Yaskawa INFORM job: A_ROOF_UPPER_0614_2_PAINT_11.JBI

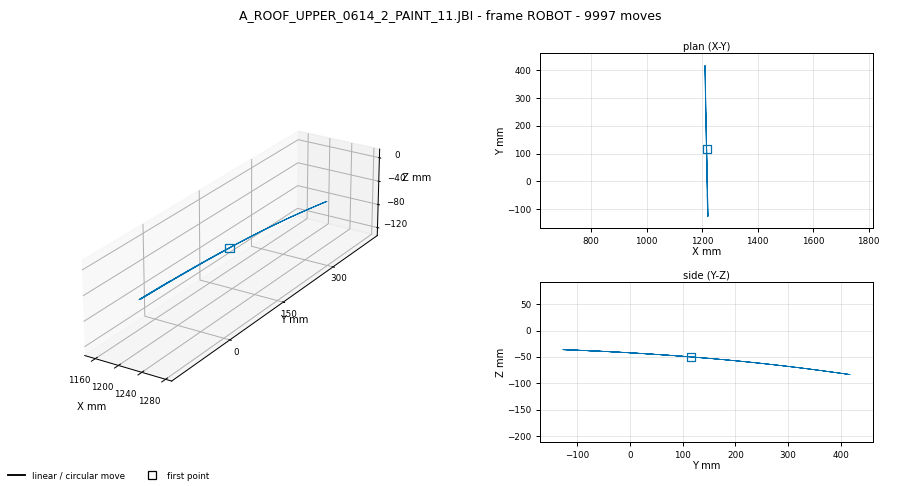
[picture p0: tool path of A_ROOF_UPPER_0614_2_PAINT_11.JBI in frame ROBOT, 9997 of 9997 moves have a stored position in this frame; points joined in program order, loops and branches not executed]
/JOB
//NAME A_ROOF_UPPER_0614_2_PAINT11
//POS
///NPOS 9997,0,0,0,0,0
///TOOL 1
///USER 0
///POSTYPE ROBOT
///RECTAN
///RCONF 1,0,0,0,0,0,0,0,0,0,0,0,0,0,0,0,0,0,0,0,0,0,0,0
C00000=1216.968,115.687,-49.725,-178.391,5.741,148.534
C00001=1216.973,115.438,-49.705,-178.393,5.741,148.535
C00002=1216.978,115.189,-49.686,-178.396,5.740,148.535
C00003=1216.982,114.939,-49.667,-178.398,5.738,148.536
C00004=1216.988,114.691,-49.647,-178.401,5.738,148.536
C00005=1216.992,114.441,-49.628,-178.403,5.737,148.537
C00006=1216.997,114.191,-49.608,-178.406,5.735,148.537
C00007=1217.002,113.943,-49.589,-178.408,5.734,148.538
C00008=1217.006,113.693,-49.570,-178.411,5.734,148.538
C00009=1217.012,113.445,-49.550,-178.414,5.732,148.539
C00010=1217.016,113.195,-49.531,-178.416,5.731,148.539
C00011=1217.020,112.946,-49.512,-178.419,5.731,148.540
C00012=1217.026,112.697,-49.492,-178.422,5.729,148.541
C00013=1217.031,112.447,-49.473,-178.424,5.728,148.541
C00014=1217.035,112.199,-49.454,-178.426,5.727,148.542
C00015=1217.040,111.949,-49.434,-178.430,5.726,148.542
C00016=1217.045,111.700,-49.415,-178.432,5.725,148.543
C00017=1217.049,111.451,-49.396,-178.434,5.724,148.543
C00018=1217.055,111.202,-49.377,-178.437,5.724,148.544
C00019=1217.060,110.952,-49.358,-178.440,5.722,148.544
C00020=1217.064,110.703,-49.339,-178.442,5.721,148.545
C00021=1217.069,110.454,-49.319,-178.444,5.720,148.545
C00022=1217.074,110.204,-49.300,-178.448,5.719,148.546
C00023=1217.078,109.956,-49.281,-178.450,5.718,148.546
C00024=1217.083,109.706,-49.261,-178.452,5.717,148.547
C00025=1217.088,109.457,-49.242,-178.455,5.716,148.547
C00026=1217.093,109.207,-49.224,-178.458,5.715,148.548
C00027=1217.098,108.959,-49.204,-178.460,5.714,148.549
C00028=1217.102,108.709,-49.185,-178.463,5.713,148.549
C00029=1217.107,108.460,-49.166,-178.466,5.712,148.550
C00030=1217.112,108.211,-49.146,-178.468,5.711,148.550
C00031=1217.117,107.962,-49.128,-178.470,5.710,148.551
C00032=1217.122,107.693,-49.107,-178.473,5.709,148.551
C00033=1217.128,107.425,-49.087,-178.476,5.708,148.552
C00034=1217.133,107.156,-49.066,-178.479,5.707,148.552
C00035=1217.138,106.888,-49.046,-178.481,5.706,148.553
C00036=1217.143,106.638,-49.027,-178.485,5.705,148.554
C00037=1217.147,106.389,-49.009,-178.487,5.704,148.554
C00038=1217.153,106.141,-48.989,-178.489,5.703,148.555
C00039=1217.157,105.891,-48.970,-178.492,5.701,148.555
C00040=1217.162,105.642,-48.952,-178.495,5.701,148.556
C00041=1217.167,105.392,-48.932,-178.497,5.700,148.556
C00042=1217.172,105.144,-48.913,-178.499,5.699,148.557
C00043=1217.177,104.893,-48.894,-178.503,5.698,148.558
C00044=1217.181,104.645,-48.876,-178.505,5.697,148.558
C00045=1217.186,104.395,-48.856,-178.507,5.696,148.559
C00046=1217.191,104.146,-48.838,-178.510,5.694,148.559
C00047=1217.195,103.898,-48.819,-178.513,5.694,148.560
C00048=1217.201,103.647,-48.800,-178.515,5.693,148.560
C00049=1217.205,103.399,-48.782,-178.517,5.692,148.561
C00050=1217.210,103.149,-48.762,-178.521,5.691,148.561
C00051=1217.215,102.900,-48.744,-178.523,5.690,148.562
C00052=1217.220,102.651,-48.724,-178.525,5.689,148.562
C00053=1217.224,102.401,-48.706,-178.528,5.689,148.563
C00054=1217.230,102.153,-48.687,-178.531,5.687,148.563
C00055=1217.234,101.903,-48.669,-178.533,5.686,148.564
C00056=1217.239,101.654,-48.649,-178.535,5.685,148.565
C00057=1217.244,101.405,-48.631,-178.538,5.685,148.565
C00058=1217.248,101.155,-48.612,-178.541,5.683,148.566
C00059=1217.254,100.906,-48.594,-178.543,5.682,148.566
C00060=1217.258,100.657,-48.575,-178.546,5.682,148.567
C00061=1217.264,100.407,-48.556,-178.549,5.680,148.568
C00062=1217.268,100.159,-48.537,-178.551,5.679,148.568
C00063=1217.273,99.909,-48.519,-178.554,5.679,148.569
C00064=1217.278,99.660,-48.500,-178.556,5.678,148.569
C00065=1217.283,99.411,-48.482,-178.559,5.676,148.570
C00066=1217.287,99.161,-48.463,-178.562,5.676,148.570
C00067=1217.292,98.912,-48.444,-178.564,5.675,148.571
C00068=1217.297,98.663,-48.426,-178.566,5.674,148.571
C00069=1217.301,98.413,-48.407,-178.569,5.672,148.572
C00070=1217.307,98.164,-48.389,-178.572,5.672,148.572
C00071=1217.312,97.915,-48.370,-178.574,5.671,148.573
C00072=1217.316,97.666,-48.352,-178.577,5.670,148.573
C00073=1217.321,97.417,-48.332,-178.579,5.670,148.574
C00074=1217.326,97.168,-48.314,-178.582,5.668,148.575
C00075=1217.331,96.918,-48.296,-178.584,5.667,148.575
C00076=1217.336,96.669,-48.277,-178.587,5.667,148.576
C00077=1217.341,96.420,-48.259,-178.589,5.666,148.576
C00078=1217.345,96.170,-48.240,-178.592,5.664,148.577
C00079=1217.350,95.921,-48.222,-178.595,5.664,148.578
C00080=1217.355,95.672,-48.203,-178.597,5.663,148.578
C00081=1217.360,95.422,-48.185,-178.600,5.662,148.579
C00082=1217.364,95.173,-48.166,-178.603,5.661,148.579
C00083=1217.370,94.924,-48.147,-178.605,5.660,148.580
C00084=1217.375,94.675,-48.129,-178.608,5.659,148.580
C00085=1217.379,94.425,-48.111,-178.610,5.659,148.581
C00086=1217.384,94.176,-48.092,-178.612,5.658,148.581
C00087=1217.389,93.927,-48.074,-178.616,5.656,148.582
C00088=1217.394,93.677,-48.056,-178.618,5.656,148.583
C00089=1217.399,93.428,-48.038,-178.620,5.655,148.583
C00090=1217.403,93.179,-48.019,-178.623,5.654,148.584
C00091=1217.408,92.930,-48.001,-178.626,5.652,148.584
C00092=1217.414,92.680,-47.982,-178.628,5.652,148.585
C00093=1217.418,92.430,-47.964,-178.631,5.651,148.585
C00094=1217.423,92.181,-47.946,-178.633,5.650,148.586
C00095=1217.428,91.933,-47.927,-178.636,5.650,148.587
C00096=1217.433,91.684,-47.909,-178.639,5.648,148.587
C00097=1217.437,91.434,-47.891,-178.641,5.647,148.588
C00098=1217.442,91.184,-47.872,-178.644,5.647,148.588
C00099=1217.447,90.935,-47.854,-178.646,5.646,148.589
C00100=1217.452,90.686,-47.836,-178.648,5.645,148.589
C00101=1217.457,90.437,-47.818,-178.652,5.644,148.590
C00102=1217.461,90.187,-47.799,-178.654,5.643,148.591
C00103=1217.466,89.938,-47.781,-178.656,5.642,148.591
C00104=1217.471,89.689,-47.763,-178.659,5.642,148.592
C00105=1217.476,89.440,-47.745,-178.662,5.641,148.592
C00106=1217.482,89.190,-47.727,-178.664,5.639,148.593
C00107=1217.486,88.941,-47.709,-178.667,5.639,148.593
C00108=1217.491,88.691,-47.691,-178.670,5.638,148.594
C00109=1217.496,88.442,-47.673,-178.672,5.637,148.594
C00110=1217.501,88.193,-47.655,-178.674,5.637,148.595
C00111=1217.506,87.944,-47.637,-178.677,5.635,148.596
C00112=1217.510,87.695,-47.619,-178.680,5.634,148.596
C00113=1217.515,87.445,-47.600,-178.682,5.634,148.597
C00114=1217.520,87.196,-47.582,-178.685,5.633,148.598
C00115=1217.525,86.946,-47.564,-178.687,5.632,148.598
C00116=1217.530,86.697,-47.546,-178.690,5.631,148.599
C00117=1217.534,86.448,-47.528,-178.693,5.630,148.599
C00118=1217.539,86.199,-47.510,-178.695,5.629,148.600
C00119=1217.544,85.949,-47.492,-178.698,5.629,148.600
C00120=1217.549,85.700,-47.474,-178.700,5.628,148.601
C00121=1217.553,85.451,-47.456,-178.702,5.627,148.601
C00122=1217.558,85.202,-47.438,-178.705,5.626,148.602
C00123=1217.563,84.952,-47.420,-178.708,5.625,148.603
C00124=1217.568,84.703,-47.402,-178.711,5.625,148.603
C00125=1217.573,84.454,-47.384,-178.713,5.624,148.604
C00126=1217.578,84.205,-47.366,-178.715,5.623,148.604
C00127=1217.583,83.956,-47.348,-178.718,5.622,148.605
C00128=1217.587,83.706,-47.330,-178.721,5.621,148.606
C00129=1217.592,83.456,-47.313,-178.723,5.620,148.606
C00130=1217.597,83.207,-47.295,-178.726,5.620,148.607
C00131=1217.602,82.958,-47.277,-178.728,5.619,148.607
C00132=1217.607,82.708,-47.259,-178.731,5.618,148.608
C00133=1217.612,82.459,-47.241,-178.733,5.617,148.609
C00134=1217.617,82.210,-47.223,-178.736,5.616,148.609
C00135=1217.622,81.960,-47.205,-178.739,5.615,148.610
C00136=1217.627,81.692,-47.186,-178.741,5.615,148.610
C00137=1217.632,81.424,-47.167,-178.744,5.614,148.611
C00138=1217.638,81.156,-47.147,-178.747,5.613,148.612
C00139=1217.643,80.887,-47.128,-178.750,5.612,148.612
C00140=1217.648,80.637,-47.111,-178.752,5.611,148.613
C00141=1217.653,80.388,-47.093,-178.755,5.610,148.613
C00142=1217.658,80.139,-47.075,-178.757,5.610,148.614
C00143=1217.663,79.889,-47.057,-178.760,5.608,148.615
C00144=1217.667,79.640,-47.040,-178.763,5.608,148.615
C00145=1217.672,79.391,-47.022,-178.765,5.607,148.616
C00146=1217.677,79.141,-47.005,-178.768,5.606,148.616
C00147=1217.682,78.892,-46.987,-178.770,5.605,148.617
C00148=1217.687,78.643,-46.969,-178.773,5.605,148.617
C00149=1217.692,78.394,-46.951,-178.775,5.604,148.618
C00150=1217.697,78.144,-46.933,-178.778,5.603,148.619
C00151=1217.701,77.895,-46.916,-178.781,5.602,148.619
C00152=1217.706,77.646,-46.898,-178.783,5.601,148.620
C00153=1217.711,77.396,-46.881,-178.786,5.601,148.620
C00154=1217.716,77.147,-46.863,-178.788,5.600,148.621
C00155=1217.721,76.898,-46.845,-178.791,5.599,148.622
C00156=1217.726,76.649,-46.828,-178.793,5.599,148.622
C00157=1217.731,76.399,-46.810,-178.796,5.598,148.623
C00158=1217.736,76.150,-46.793,-178.798,5.596,148.623
C00159=1217.741,75.900,-46.775,-178.801,5.596,148.624
C00160=1217.746,75.651,-46.757,-178.804,5.595,148.625
C00161=1217.750,75.402,-46.740,-178.806,5.595,148.625
C00162=1217.755,75.153,-46.722,-178.809,5.594,148.626
C00163=1217.760,74.903,-46.705,-178.811,5.593,148.626
C00164=1217.765,74.654,-46.687,-178.814,5.593,148.627
C00165=1217.770,74.404,-46.670,-178.816,5.592,148.627
C00166=1217.775,74.155,-46.652,-178.819,5.590,148.628
C00167=1217.779,73.906,-46.634,-178.822,5.590,148.629
C00168=1217.785,73.656,-46.617,-178.824,5.589,148.629
C00169=1217.789,73.407,-46.600,-178.826,5.588,148.630
C00170=1217.794,73.157,-46.583,-178.829,5.588,148.631
C00171=1217.800,72.909,-46.565,-178.832,5.587,148.631
C00172=1217.804,72.659,-46.548,-178.834,5.586,148.632
C00173=1217.809,72.410,-46.530,-178.837,5.585,148.632
C00174=1217.814,72.160,-46.513,-178.839,5.585,148.633
C00175=1217.819,71.911,-46.496,-178.842,5.584,148.634
C00176=1217.824,71.662,-46.478,-178.845,5.583,148.634
C00177=1217.829,71.412,-46.461,-178.847,5.582,148.635
C00178=1217.833,71.163,-46.444,-178.850,5.581,148.635
C00179=1217.838,70.913,-46.426,-178.852,5.581,148.636
C00180=1217.843,70.664,-46.408,-178.855,5.580,148.637
C00181=1217.848,70.415,-46.392,-178.857,5.579,148.637
C00182=1217.853,70.165,-46.375,-178.860,5.579,148.638
C00183=1217.858,69.916,-46.357,-178.862,5.578,148.638
C00184=1217.863,69.667,-46.340,-178.865,5.578,148.639
C00185=1217.868,69.418,-46.322,-178.867,5.577,148.640
C00186=1217.873,69.168,-46.305,-178.870,5.575,148.640
C00187=1217.877,68.918,-46.288,-178.873,5.575,148.641
C00188=1217.882,68.669,-46.270,-178.876,5.574,148.641
C00189=1217.887,68.420,-46.254,-178.878,5.573,148.642
C00190=1217.893,68.171,-46.237,-178.880,5.573,148.643
C00191=1217.897,67.922,-46.219,-178.883,5.572,148.643
C00192=1217.902,67.672,-46.202,-178.886,5.572,148.644
C00193=1217.907,67.422,-46.185,-178.888,5.571,148.644
C00194=1217.911,67.173,-46.168,-178.890,5.570,148.645
C00195=1217.917,66.923,-46.150,-178.893,5.569,148.646
C00196=1217.922,66.675,-46.134,-178.896,5.569,148.646
C00197=1217.927,66.426,-46.116,-178.898,5.568,148.647
C00198=1217.931,66.176,-46.099,-178.901,5.567,148.647
C00199=1217.936,65.926,-46.082,-178.904,5.566,148.648
C00200=1217.941,65.677,-46.065,-178.906,5.565,148.649
C00201=1217.946,65.428,-46.047,-178.909,5.565,148.649
C00202=1217.951,65.179,-46.031,-178.911,5.564,148.650
C00203=1217.956,64.929,-46.014,-178.914,5.563,148.650
C00204=1217.961,64.680,-45.997,-178.916,5.563,148.651
C00205=1217.966,64.430,-45.980,-178.919,5.562,148.652
C00206=1217.970,64.181,-45.962,-178.921,5.561,148.652
C00207=1217.976,63.932,-45.946,-178.924,5.561,148.653
C00208=1217.980,63.682,-45.929,-178.926,5.560,148.654
C00209=1217.985,63.432,-45.912,-178.929,5.560,148.654
C00210=1217.990,63.183,-45.895,-178.931,5.559,148.655
C00211=1217.996,62.934,-45.878,-178.934,5.558,148.655
C00212=1218.000,62.685,-45.861,-178.936,5.558,148.656
C00213=1218.005,62.435,-45.843,-178.939,5.557,148.657
C00214=1218.010,62.186,-45.827,-178.942,5.556,148.657
C00215=1218.015,61.936,-45.810,-178.944,5.555,148.658
C00216=1218.020,61.687,-45.793,-178.947,5.554,148.658
C00217=1218.024,61.438,-45.777,-178.950,5.554,148.659
C00218=1218.030,61.188,-45.759,-178.952,5.553,148.660
C00219=1218.034,60.938,-45.743,-178.955,5.552,148.660
C00220=1218.040,60.689,-45.726,-178.957,5.551,148.661
C00221=1218.044,60.440,-45.709,-178.960,5.551,148.662
C00222=1218.049,60.191,-45.691,-178.962,5.550,148.662
C00223=1218.054,59.942,-45.675,-178.965,5.550,148.663
C00224=1218.059,59.692,-45.658,-178.967,5.549,148.663
C00225=1218.064,59.443,-45.641,-178.970,5.548,148.664
C00226=1218.069,59.193,-45.624,-178.972,5.548,148.665
C00227=1218.074,58.944,-45.608,-178.975,5.547,148.665
C00228=1218.079,58.695,-45.591,-178.978,5.547,148.666
C00229=1218.083,58.445,-45.574,-178.980,5.546,148.666
C00230=1218.089,58.196,-45.557,-178.982,5.545,148.667
C00231=1218.094,57.946,-45.540,-178.985,5.545,148.668
C00232=1218.098,57.697,-45.524,-178.988,5.544,148.668
C00233=1218.104,57.448,-45.507,-178.990,5.543,148.669
C00234=1218.108,57.198,-45.490,-178.992,5.543,148.670
C00235=1218.113,56.948,-45.474,-178.995,5.542,148.670
C00236=1218.118,56.699,-45.457,-178.998,5.541,148.671
C00237=1218.123,56.450,-45.441,-179.000,5.541,148.672
C00238=1218.128,56.200,-45.424,-179.003,5.540,148.672
C00239=1218.132,55.951,-45.407,-179.005,5.539,148.673
C00240=1218.138,55.683,-45.389,-179.008,5.538,148.673
C00241=1218.144,55.415,-45.371,-179.011,5.537,148.674
C00242=1218.149,55.146,-45.354,-179.014,5.537,148.675
C00243=1218.155,54.877,-45.335,-179.016,5.536,148.675
C00244=1218.159,54.628,-45.319,-179.019,5.536,148.676
C00245=1218.164,54.378,-45.302,-179.022,5.535,148.677
C00246=1218.169,54.129,-45.285,-179.024,5.535,148.677
C00247=1218.174,53.879,-45.269,-179.027,5.534,148.678
C00248=1218.179,53.630,-45.253,-179.029,5.533,148.679
C00249=1218.184,53.381,-45.236,-179.032,5.533,148.679
C00250=1218.189,53.131,-45.219,-179.034,5.532,148.680
C00251=1218.194,52.882,-45.203,-179.037,5.531,148.680
C00252=1218.199,52.633,-45.186,-179.039,5.531,148.681
C00253=1218.203,52.383,-45.170,-179.042,5.530,148.682
C00254=1218.208,52.134,-45.154,-179.044,5.529,148.682
C00255=1218.214,51.884,-45.137,-179.047,5.529,148.683
C00256=1218.219,51.635,-45.120,-179.050,5.528,148.683
C00257=1218.223,51.385,-45.104,-179.052,5.528,148.684
C00258=1218.228,51.136,-45.088,-179.055,5.527,148.685
C00259=1218.233,50.887,-45.071,-179.057,5.527,148.686
C00260=1218.238,50.638,-45.055,-179.060,5.526,148.686
C00261=1218.244,50.388,-45.038,-179.062,5.525,148.687
C00262=1218.248,50.138,-45.022,-179.065,5.525,148.687
C00263=1218.253,49.889,-45.005,-179.067,5.524,148.688
C00264=1218.258,49.639,-44.990,-179.070,5.523,148.689
C00265=1218.262,49.390,-44.973,-179.072,5.523,148.689
C00266=1218.268,49.141,-44.957,-179.075,5.522,148.690
C00267=1218.272,48.892,-44.940,-179.078,5.521,148.690
C00268=1218.278,48.642,-44.924,-179.080,5.521,148.691
C00269=1218.283,48.393,-44.907,-179.083,5.520,148.692
C00270=1218.288,48.144,-44.891,-179.085,5.520,148.692
C00271=1218.293,47.894,-44.875,-179.088,5.519,148.693
C00272=1218.297,47.644,-44.858,-179.090,5.518,148.694
C00273=1218.302,47.395,-44.843,-179.093,5.518,148.694
C00274=1218.307,47.145,-44.826,-179.096,5.517,148.695
C00275=1218.312,46.897,-44.810,-179.098,5.517,148.696
C00276=1218.317,46.646,-44.794,-179.101,5.516,148.696
C00277=1218.322,46.398,-44.777,-179.103,5.515,148.697
C00278=1218.327,46.148,-44.761,-179.106,5.515,148.697
C00279=1218.332,45.898,-44.744,-179.108,5.514,148.698
C00280=1218.337,45.649,-44.728,-179.111,5.514,148.699
C00281=1218.342,45.400,-44.712,-179.114,5.513,148.699
C00282=1218.347,45.150,-44.696,-179.116,5.512,148.700
C00283=1218.352,44.901,-44.680,-179.118,5.512,148.700
C00284=1218.357,44.651,-44.663,-179.121,5.511,148.701
C00285=1218.362,44.402,-44.648,-179.124,5.510,148.702
C00286=1218.366,44.152,-44.631,-179.126,5.510,148.702
C00287=1218.372,43.903,-44.615,-179.129,5.509,148.703
C00288=1218.376,43.653,-44.599,-179.131,5.509,148.704
C00289=1218.382,43.404,-44.583,-179.134,5.508,148.704
C00290=1218.386,43.155,-44.567,-179.136,5.507,148.705
C00291=1218.392,42.905,-44.551,-179.139,5.507,148.706
C00292=1218.397,42.656,-44.535,-179.141,5.507,148.706
C00293=1218.401,42.406,-44.519,-179.144,5.506,148.707
C00294=1218.407,42.157,-44.503,-179.146,5.506,148.708
C00295=1218.411,41.907,-44.486,-179.149,5.505,148.708
C00296=1218.417,41.658,-44.471,-179.151,5.504,148.709
C00297=1218.421,41.408,-44.454,-179.154,5.504,148.709
C00298=1218.427,41.159,-44.439,-179.156,5.503,148.710
C00299=1218.430,40.910,-44.422,-179.159,5.503,148.711
C00300=1218.436,40.660,-44.407,-179.162,5.502,148.711
C00301=1218.441,40.411,-44.391,-179.164,5.502,148.712
C00302=1218.446,40.162,-44.375,-179.167,5.501,148.713
C00303=1218.451,39.912,-44.359,-179.169,5.500,148.713
C00304=1218.456,39.662,-44.343,-179.172,5.500,148.714
C00305=1218.461,39.413,-44.327,-179.174,5.499,148.715
C00306=1218.466,39.164,-44.311,-179.177,5.499,148.715
C00307=1218.471,38.914,-44.295,-179.180,5.498,148.716
C00308=1218.476,38.665,-44.279,-179.182,5.498,148.717
C00309=1218.481,38.415,-44.263,-179.185,5.497,148.717
C00310=1218.486,38.166,-44.248,-179.187,5.496,148.718
C00311=1218.491,37.917,-44.232,-179.189,5.496,148.718
C00312=1218.495,37.667,-44.216,-179.192,5.496,148.719
C00313=1218.501,37.418,-44.200,-179.194,5.495,148.720
C00314=1218.505,37.168,-44.183,-179.197,5.495,148.720
C00315=1218.511,36.919,-44.168,-179.200,5.494,148.721
C00316=1218.516,36.669,-44.152,-179.202,5.494,148.722
C00317=1218.520,36.419,-44.137,-179.205,5.493,148.722
C00318=1218.525,36.171,-44.121,-179.207,5.492,148.723
C00319=1218.531,35.921,-44.105,-179.210,5.492,148.724
C00320=1218.535,35.671,-44.089,-179.212,5.491,148.724
C00321=1218.541,35.422,-44.074,-179.215,5.491,148.725
C00322=1218.546,35.173,-44.057,-179.218,5.490,148.726
C00323=1218.550,34.923,-44.042,-179.220,5.489,148.726
C00324=1218.555,34.674,-44.026,-179.223,5.489,148.727
C00325=1218.561,34.424,-44.011,-179.225,5.489,148.727
C00326=1218.565,34.174,-43.995,-179.227,5.488,148.728
C00327=1218.571,33.925,-43.979,-179.230,5.488,148.729
C00328=1218.575,33.676,-43.963,-179.232,5.487,148.729
C00329=1218.580,33.426,-43.947,-179.235,5.487,148.730
C00330=1218.585,33.177,-43.932,-179.238,5.486,148.731
C00331=1218.591,32.927,-43.916,-179.240,5.486,148.731
C00332=1218.595,32.678,-43.901,-179.243,5.485,148.732
C00333=1218.600,32.428,-43.885,-179.245,5.484,148.733
C00334=1218.606,32.179,-43.870,-179.248,5.484,148.733
C00335=1218.610,31.929,-43.853,-179.250,5.483,148.734
C00336=1218.615,31.680,-43.838,-179.253,5.483,148.735
C00337=1218.620,31.431,-43.823,-179.255,5.483,148.735
C00338=1218.625,31.182,-43.807,-179.258,5.482,148.736
C00339=1218.629,30.932,-43.792,-179.260,5.482,148.737
C00340=1218.635,30.682,-43.776,-179.263,5.481,148.737
C00341=1218.640,30.433,-43.760,-179.266,5.481,148.738
C00342=1218.644,30.183,-43.745,-179.268,5.480,148.738
C00343=1218.650,29.934,-43.729,-179.271,5.479,148.739
C00344=1218.655,29.665,-43.712,-179.273,5.479,148.740
C00345=1218.661,29.397,-43.695,-179.276,5.478,148.741
C00346=1218.666,29.128,-43.680,-179.279,5.478,148.741
C00347=1218.671,28.859,-43.663,-179.282,5.477,148.742
C00348=1218.676,28.609,-43.647,-179.284,5.477,148.743
C00349=1218.681,28.360,-43.632,-179.286,5.476,148.743
C00350=1218.686,28.111,-43.616,-179.289,5.475,148.744
C00351=1218.692,27.861,-43.601,-179.292,5.475,148.745
C00352=1218.696,27.612,-43.586,-179.294,5.475,148.745
C00353=1218.701,27.362,-43.570,-179.296,5.475,148.746
C00354=1218.707,27.113,-43.554,-179.299,5.474,148.747
C00355=1218.711,26.864,-43.539,-179.302,5.473,148.747
C00356=1218.717,26.614,-43.523,-179.304,5.473,148.748
C00357=1218.721,26.365,-43.508,-179.307,5.472,148.749
C00358=1218.726,26.115,-43.493,-179.310,5.472,148.749
C00359=1218.732,25.865,-43.478,-179.312,5.471,148.750
C00360=1218.736,25.616,-43.463,-179.314,5.470,148.750
C00361=1218.742,25.367,-43.447,-179.317,5.471,148.751
C00362=1218.746,25.117,-43.432,-179.319,5.470,148.752
C00363=1218.751,24.867,-43.416,-179.322,5.470,148.752
C00364=1218.756,24.618,-43.401,-179.324,5.469,148.753
C00365=1218.761,24.369,-43.386,-179.327,5.469,148.754
C00366=1218.767,24.119,-43.371,-179.330,5.468,148.755
C00367=1218.771,23.869,-43.355,-179.332,5.468,148.755
C00368=1218.776,23.620,-43.340,-179.335,5.467,148.756
C00369=1218.781,23.371,-43.325,-179.337,5.467,148.756
C00370=1218.786,23.121,-43.309,-179.339,5.466,148.757
C00371=1218.791,22.872,-43.294,-179.342,5.466,148.758
C00372=1218.797,22.622,-43.279,-179.345,5.465,148.758
C00373=1218.801,22.372,-43.264,-179.347,5.465,148.759
C00374=1218.806,22.123,-43.248,-179.350,5.464,148.760
C00375=1218.811,21.874,-43.233,-179.352,5.464,148.760
C00376=1218.816,21.624,-43.218,-179.355,5.464,148.761
C00377=1218.821,21.375,-43.203,-179.357,5.463,148.762
C00378=1218.827,21.125,-43.188,-179.360,5.463,148.762
C00379=1218.831,20.876,-43.173,-179.362,5.462,148.763
C00380=1218.837,20.626,-43.158,-179.365,5.461,148.764
C00381=1218.841,20.376,-43.143,-179.367,5.461,148.764
C00382=1218.846,20.127,-43.127,-179.370,5.460,148.765
C00383=1218.851,19.878,-43.112,-179.372,5.461,148.766
C00384=1218.856,19.628,-43.098,-179.375,5.460,148.766
C00385=1218.861,19.379,-43.082,-179.377,5.460,148.767
C00386=1218.866,19.130,-43.067,-179.380,5.459,148.768
C00387=1218.872,18.880,-43.052,-179.383,5.459,148.768
C00388=1218.876,18.631,-43.037,-179.385,5.458,148.769
C00389=1218.882,18.381,-43.022,-179.388,5.458,148.770
C00390=1218.886,18.131,-43.007,-179.389,5.457,148.770
C00391=1218.891,17.882,-42.992,-179.392,5.457,148.771
C00392=1218.896,17.632,-42.977,-179.395,5.456,148.772
C00393=1218.901,17.383,-42.962,-179.397,5.456,148.772
C00394=1218.906,17.133,-42.947,-179.400,5.455,148.773
C00395=1218.911,16.884,-42.932,-179.403,5.455,148.774
C00396=1218.916,16.634,-42.917,-179.405,5.454,148.774
C00397=1218.921,16.385,-42.902,-179.407,5.455,148.775
C00398=1218.926,16.135,-42.888,-179.410,5.454,148.776
C00399=1218.932,15.886,-42.872,-179.413,5.453,148.776
C00400=1218.936,15.637,-42.857,-179.415,5.453,148.777
C00401=1218.941,15.387,-42.843,-179.418,5.452,148.778
C00402=1218.947,15.138,-42.827,-179.420,5.452,148.778
C00403=1218.952,14.888,-42.813,-179.422,5.452,148.779
C00404=1218.956,14.639,-42.798,-179.425,5.451,148.780
C00405=1218.962,14.389,-42.783,-179.428,5.451,148.780
C00406=1218.966,14.139,-42.768,-179.430,5.450,148.781
C00407=1218.971,13.889,-42.753,-179.433,5.450,148.782
C00408=1218.976,13.640,-42.738,-179.436,5.449,148.782
C00409=1218.981,13.390,-42.723,-179.438,5.449,148.783
C00410=1218.986,13.141,-42.708,-179.440,5.449,148.784
C00411=1218.991,12.891,-42.694,-179.443,5.448,148.784
C00412=1218.996,12.642,-42.679,-179.446,5.448,148.785
C00413=1219.001,12.392,-42.664,-179.448,5.447,148.786
C00414=1219.006,12.143,-42.649,-179.451,5.447,148.786
C00415=1219.012,11.893,-42.634,-179.452,5.447,148.787
C00416=1219.016,11.644,-42.619,-179.455,5.446,148.787
C00417=1219.021,11.394,-42.605,-179.458,5.446,148.788
C00418=1219.026,11.145,-42.590,-179.460,5.445,148.789
C00419=1219.032,10.895,-42.575,-179.463,5.445,148.790
C00420=1219.037,10.646,-42.561,-179.465,5.445,148.790
C00421=1219.041,10.397,-42.546,-179.468,5.444,148.791
C00422=1219.047,10.148,-42.532,-179.470,5.444,148.792
C00423=1219.052,9.898,-42.517,-179.473,5.443,148.792
C00424=1219.057,9.648,-42.502,-179.476,5.443,148.793
C00425=1219.062,9.399,-42.488,-179.478,5.443,148.794
C00426=1219.067,9.150,-42.473,-179.480,5.443,148.794
C00427=1219.072,8.900,-42.459,-179.483,5.442,148.795
C00428=1219.077,8.650,-42.444,-179.486,5.442,148.796
C00429=1219.082,8.401,-42.429,-179.488,5.441,148.796
C00430=1219.087,8.151,-42.415,-179.491,5.440,148.797
C00431=1219.092,7.901,-42.400,-179.493,5.440,148.798
C00432=1219.097,7.652,-42.385,-179.495,5.440,148.798
C00433=1219.102,7.402,-42.370,-179.498,5.439,148.799
C00434=1219.107,7.153,-42.356,-179.501,5.439,148.800
C00435=1219.112,6.903,-42.341,-179.503,5.438,148.800
C00436=1219.117,6.654,-42.327,-179.505,5.439,148.801
C00437=1219.122,6.404,-42.313,-179.508,5.438,148.802
C00438=1219.127,6.154,-42.298,-179.511,5.438,148.802
C00439=1219.132,5.906,-42.284,-179.513,5.437,148.803
C00440=1219.138,5.656,-42.269,-179.516,5.437,148.804
C00441=1219.143,5.406,-42.255,-179.518,5.437,148.804
C00442=1219.148,5.156,-42.240,-179.521,5.436,148.805
C00443=1219.152,4.907,-42.225,-179.523,5.436,148.806
C00444=1219.157,4.658,-42.211,-179.526,5.435,148.806
C00445=1219.162,4.408,-42.197,-179.528,5.434,148.807
C00446=1219.167,4.158,-42.182,-179.530,5.435,148.808
C00447=1219.172,3.909,-42.167,-179.533,5.434,148.808
C00448=1219.178,3.639,-42.152,-179.536,5.434,148.809
C00449=1219.184,3.371,-42.137,-179.539,5.434,148.810
C00450=1219.189,3.103,-42.121,-179.541,5.433,148.811
C00451=1219.194,2.833,-42.106,-179.544,5.433,148.811
C00452=1219.199,2.583,-42.092,-179.547,5.432,148.812
C00453=1219.204,2.334,-42.077,-179.549,5.432,148.813
C00454=1219.209,2.085,-42.062,-179.551,5.432,148.813
C00455=1219.214,1.835,-42.048,-179.554,5.431,148.814
C00456=1219.219,1.586,-42.034,-179.557,5.431,148.815
C00457=1219.224,1.336,-42.020,-179.559,5.430,148.815
C00458=1219.229,1.086,-42.006,-179.561,5.431,148.816
C00459=1219.234,0.837,-41.991,-179.564,5.430,148.817
C00460=1219.240,0.587,-41.976,-179.567,5.430,148.817
C00461=1219.244,0.338,-41.961,-179.569,5.429,148.818
C00462=1219.250,0.089,-41.947,-179.571,5.429,148.819
C00463=1219.255,-0.161,-41.933,-179.574,5.428,148.819
C00464=1219.260,-0.411,-41.919,-179.576,5.428,148.820
C00465=1219.265,-0.660,-41.905,-179.579,5.427,148.821
C00466=1219.270,-0.910,-41.890,-179.581,5.427,148.821
C00467=1219.275,-1.160,-41.876,-179.584,5.427,148.822
C00468=1219.280,-1.409,-41.862,-179.586,5.427,148.823
C00469=1219.285,-1.658,-41.849,-179.589,5.426,148.823
C00470=1219.290,-1.908,-41.834,-179.592,5.426,148.824
C00471=1219.294,-2.158,-41.820,-179.594,5.426,148.825
C00472=1219.299,-2.407,-41.806,-179.596,5.425,148.826
C00473=1219.305,-2.656,-41.792,-179.599,5.425,148.826
C00474=1219.310,-2.906,-41.777,-179.602,5.424,148.827
C00475=1219.315,-3.156,-41.763,-179.604,5.425,148.828
C00476=1219.320,-3.406,-41.749,-179.606,5.424,148.828
C00477=1219.325,-3.655,-41.735,-179.609,5.424,148.829
C00478=1219.330,-3.904,-41.721,-179.612,5.423,148.830
C00479=1219.335,-4.154,-41.706,-179.614,5.423,148.830
C00480=1219.340,-4.404,-41.692,-179.616,5.423,148.831
C00481=1219.346,-4.653,-41.678,-179.618,5.422,148.831
C00482=1219.351,-4.902,-41.664,-179.621,5.422,148.832
C00483=1219.356,-5.152,-41.650,-179.623,5.422,148.833
C00484=1219.360,-5.402,-41.637,-179.626,5.421,148.834
C00485=1219.366,-5.651,-41.623,-179.629,5.421,148.834
C00486=1219.371,-5.901,-41.609,-179.631,5.420,148.835
C00487=1219.376,-6.151,-41.594,-179.633,5.421,148.836
C00488=1219.381,-6.400,-41.580,-179.636,5.420,148.836
C00489=1219.386,-6.649,-41.566,-179.639,5.420,148.837
C00490=1219.391,-6.899,-41.552,-179.641,5.419,148.838
C00491=1219.395,-7.148,-41.538,-179.643,5.419,148.838
C00492=1219.401,-7.399,-41.525,-179.646,5.419,148.839
C00493=1219.406,-7.648,-41.511,-179.649,5.418,148.840
C00494=1219.411,-7.897,-41.496,-179.651,5.418,148.840
C00495=1219.416,-8.147,-41.482,-179.653,5.418,148.841
C00496=1219.422,-8.396,-41.468,-179.656,5.418,148.842
C00497=1219.426,-8.646,-41.455,-179.659,5.417,148.843
C00498=1219.431,-8.896,-41.441,-179.661,5.417,148.843
C00499=1219.437,-9.145,-41.427,-179.663,5.417,148.844
C00500=1219.442,-9.395,-41.413,-179.666,5.416,148.845
C00501=1219.447,-9.644,-41.399,-179.669,5.416,148.845
C00502=1219.451,-9.894,-41.385,-179.671,5.415,148.846
C00503=1219.457,-10.143,-41.372,-179.673,5.415,148.846
C00504=1219.462,-10.393,-41.357,-179.676,5.415,148.847
C00505=1219.467,-10.643,-41.343,-179.678,5.414,148.848
C00506=1219.471,-10.891,-41.330,-179.681,5.414,148.849
C00507=1219.477,-11.142,-41.316,-179.683,5.414,148.849
C00508=1219.482,-11.392,-41.302,-179.686,5.414,148.850
C00509=1219.487,-11.641,-41.288,-179.688,5.413,148.851
C00510=1219.492,-11.891,-41.274,-179.691,5.413,148.851
C00511=1219.497,-12.140,-41.261,-179.693,5.413,148.852
C00512=1219.502,-12.389,-41.247,-179.696,5.412,148.853
C00513=1219.507,-12.640,-41.233,-179.698,5.412,148.853
C00514=1219.512,-12.888,-41.220,-179.700,5.412,148.854
C00515=1219.517,-13.138,-41.206,-179.703,5.412,148.855
C00516=1219.522,-13.388,-41.191,-179.706,5.411,148.855
C00517=1219.528,-13.637,-41.178,-179.708,5.411,148.856
C00518=1219.532,-13.887,-41.165,-179.710,5.411,148.857
C00519=1219.538,-14.137,-41.151,-179.713,5.411,148.858
C00520=1219.543,-14.386,-41.137,-179.716,5.410,148.858
C00521=1219.547,-14.636,-41.123,-179.718,5.410,148.859
C00522=1219.553,-14.885,-41.110,-179.721,5.410,148.860
C00523=1219.558,-15.135,-41.096,-179.723,5.409,148.860
C00524=1219.562,-15.384,-41.082,-179.726,5.409,148.861
C00525=1219.568,-15.634,-41.069,-179.728,5.409,148.862
C00526=1219.573,-15.884,-41.055,-179.731,5.409,148.862
C00527=1219.578,-16.133,-41.042,-179.733,5.408,148.863
C00528=1219.583,-16.383,-41.028,-179.736,5.408,148.864
C00529=1219.589,-16.633,-41.014,-179.738,5.408,148.865
C00530=1219.593,-16.882,-41.001,-179.740,5.407,148.865
C00531=1219.598,-17.131,-40.987,-179.743,5.407,148.866
C00532=1219.604,-17.381,-40.974,-179.745,5.407,148.866
C00533=1219.608,-17.630,-40.960,-179.748,5.406,148.867
C00534=1219.614,-17.880,-40.947,-179.750,5.406,148.868
C00535=1219.618,-18.129,-40.933,-179.753,5.405,148.868
C00536=1219.624,-18.380,-40.919,-179.755,5.406,148.869
C00537=1219.629,-18.629,-40.905,-179.758,5.405,148.870
C00538=1219.634,-18.879,-40.893,-179.760,5.405,148.871
C00539=1219.639,-19.128,-40.879,-179.762,5.405,148.871
C00540=1219.644,-19.378,-40.866,-179.765,5.405,148.872
C00541=1219.649,-19.627,-40.852,-179.768,5.404,148.873
C00542=1219.655,-19.877,-40.838,-179.770,5.404,148.873
C00543=1219.659,-20.126,-40.825,-179.772,5.404,148.874
C00544=1219.665,-20.376,-40.811,-179.775,5.403,148.875
C00545=1219.670,-20.625,-40.799,-179.778,5.403,148.875
C00546=1219.675,-20.875,-40.784,-179.780,5.403,148.876
C00547=1219.680,-21.125,-40.772,-179.782,5.403,148.877
C00548=1219.685,-21.374,-40.758,-179.785,5.402,148.877
C00549=1219.691,-21.624,-40.744,-179.787,5.403,148.878
C00550=1219.695,-21.873,-40.731,-179.790,5.402,148.879
C00551=1219.701,-22.123,-40.717,-179.792,5.402,148.880
C00552=1219.706,-22.392,-40.703,-179.795,5.401,148.880
C00553=1219.711,-22.662,-40.689,-179.797,5.401,148.881
C00554=1219.717,-22.931,-40.674,-179.800,5.401,148.882
C00555=1219.722,-23.200,-40.660,-179.803,5.401,148.883
C00556=1219.727,-23.450,-40.646,-179.806,5.400,148.883
C00557=1219.732,-23.699,-40.634,-179.808,5.401,148.884
C00558=1219.738,-23.950,-40.620,-179.810,5.400,148.885
C00559=1219.742,-24.199,-40.607,-179.813,5.399,148.885
C00560=1219.748,-24.449,-40.593,-179.815,5.400,148.886
C00561=1219.753,-24.698,-40.581,-179.817,5.399,148.887
C00562=1219.758,-24.948,-40.566,-179.820,5.399,148.887
C00563=1219.763,-25.197,-40.554,-179.823,5.398,148.888
C00564=1219.768,-25.448,-40.540,-179.825,5.398,148.889
C00565=1219.773,-25.696,-40.527,-179.827,5.398,148.889
C00566=1219.778,-25.946,-40.514,-179.830,5.397,148.890
C00567=1219.783,-26.196,-40.501,-179.832,5.398,148.891
C00568=1219.789,-26.445,-40.488,-179.835,5.397,148.891
C00569=1219.793,-26.695,-40.474,-179.837,5.397,148.892
C00570=1219.799,-26.944,-40.461,-179.840,5.397,148.893
C00571=1219.804,-27.195,-40.448,-179.842,5.397,148.893
C00572=1219.809,-27.444,-40.435,-179.845,5.396,148.894
C00573=1219.813,-27.693,-40.421,-179.847,5.396,148.895
C00574=1219.819,-27.943,-40.408,-179.850,5.396,148.896
C00575=1219.824,-28.193,-40.395,-179.852,5.395,148.896
C00576=1219.829,-28.443,-40.382,-179.854,5.396,148.897
C00577=1219.835,-28.692,-40.369,-179.857,5.395,148.898
C00578=1219.839,-28.941,-40.356,-179.860,5.395,148.898
C00579=1219.845,-29.191,-40.342,-179.862,5.395,148.899
C00580=1219.849,-29.441,-40.330,-179.864,5.395,148.900
C00581=1219.854,-29.690,-40.317,-179.867,5.394,148.900
C00582=1219.860,-29.940,-40.304,-179.869,5.394,148.901
C00583=1219.864,-30.189,-40.290,-179.872,5.394,148.902
C00584=1219.870,-30.439,-40.277,-179.874,5.393,148.903
C00585=1219.875,-30.689,-40.264,-179.877,5.394,148.903
C00586=1219.880,-30.938,-40.251,-179.879,5.393,148.904
C00587=1219.885,-31.188,-40.239,-179.882,5.393,148.905
C00588=1219.890,-31.438,-40.225,-179.884,5.393,148.905
C00589=1219.895,-31.687,-40.213,-179.887,5.393,148.906
C00590=1219.901,-31.936,-40.200,-179.889,5.392,148.907
C00591=1219.906,-32.187,-40.186,-179.891,5.392,148.907
C00592=1219.911,-32.436,-40.173,-179.894,5.392,148.908
C00593=1219.916,-32.685,-40.160,-179.897,5.391,148.909
C00594=1219.921,-32.935,-40.147,-179.898,5.391,148.909
C00595=1219.926,-33.184,-40.134,-179.901,5.391,148.910
C00596=1219.931,-33.435,-40.121,-179.904,5.390,148.911
C00597=1219.937,-33.684,-40.108,-179.906,5.391,148.911
C00598=1219.942,-33.933,-40.096,-179.908,5.390,148.912
C00599=1219.946,-34.183,-40.083,-179.911,5.390,148.913
C00600=1219.951,-34.433,-40.070,-179.913,5.390,148.914
C00601=1219.957,-34.682,-40.057,-179.916,5.390,148.914
C00602=1219.962,-34.932,-40.044,-179.918,5.389,148.915
C00603=1219.967,-35.182,-40.031,-179.920,5.389,148.916
C00604=1219.972,-35.431,-40.019,-179.923,5.389,148.916
C00605=1219.978,-35.681,-40.005,-179.925,5.389,148.917
C00606=1219.982,-35.931,-39.992,-179.928,5.389,148.918
C00607=1219.987,-36.180,-39.980,-179.931,5.388,148.918
C00608=1219.993,-36.429,-39.967,-179.933,5.389,148.919
C00609=1219.997,-36.679,-39.954,-179.935,5.388,148.920
C00610=1220.003,-36.929,-39.941,-179.938,5.388,148.920
C00611=1220.008,-37.178,-39.928,-179.940,5.388,148.921
C00612=1220.013,-37.428,-39.915,-179.943,5.388,148.922
C00613=1220.018,-37.678,-39.903,-179.945,5.387,148.923
C00614=1220.024,-37.927,-39.890,-179.947,5.387,148.923
C00615=1220.029,-38.177,-39.877,-179.950,5.387,148.924
C00616=1220.034,-38.427,-39.865,-179.953,5.386,148.925
C00617=1220.039,-38.677,-39.852,-179.955,5.387,148.925
C00618=1220.044,-38.926,-39.840,-179.958,5.386,148.926
C00619=1220.049,-39.175,-39.827,-179.960,5.386,148.927
C00620=1220.054,-39.426,-39.813,-179.962,5.386,148.927
C00621=1220.059,-39.675,-39.801,-179.965,5.386,148.928
C00622=1220.064,-39.924,-39.788,-179.967,5.386,148.929
C00623=1220.070,-40.173,-39.776,-179.970,5.385,148.930
C00624=1220.074,-40.424,-39.763,-179.972,5.385,148.930
C00625=1220.079,-40.673,-39.751,-179.974,5.385,148.931
C00626=1220.085,-40.923,-39.738,-179.977,5.385,148.932
C00627=1220.090,-41.172,-39.726,-179.980,5.384,148.932
C00628=1220.095,-41.422,-39.712,-179.982,5.385,148.933
C00629=1220.100,-41.672,-39.699,-179.984,5.384,148.934
C00630=1220.106,-41.922,-39.688,-179.986,5.384,148.934
C00631=1220.111,-42.171,-39.675,-179.989,5.384,148.935
C00632=1220.115,-42.421,-39.662,-179.991,5.383,148.936
C00633=1220.120,-42.670,-39.649,-179.994,5.384,148.936
C00634=1220.125,-42.920,-39.637,-179.996,5.383,148.937
C00635=1220.131,-43.170,-39.625,-179.999,5.383,148.938
C00636=1220.136,-43.419,-39.612,179.999,5.383,148.938
C00637=1220.140,-43.669,-39.599,179.996,5.382,148.939
C00638=1220.146,-43.918,-39.587,179.994,5.383,148.940
C00639=1220.152,-44.168,-39.574,179.992,5.382,148.941
C00640=1220.157,-44.418,-39.562,179.989,5.382,148.941
C00641=1220.162,-44.667,-39.549,179.987,5.382,148.942
C00642=1220.167,-44.917,-39.536,179.984,5.382,148.943
C00643=1220.172,-45.167,-39.524,179.982,5.381,148.943
C00644=1220.177,-45.416,-39.512,179.979,5.381,148.944
C00645=1220.182,-45.666,-39.499,179.977,5.381,148.945
C00646=1220.188,-45.916,-39.487,179.975,5.381,148.945
C00647=1220.193,-46.165,-39.475,179.972,5.381,148.946
C00648=1220.197,-46.415,-39.462,179.969,5.380,148.947
C00649=1220.203,-46.665,-39.450,179.967,5.381,148.948
C00650=1220.208,-46.914,-39.437,179.965,5.380,148.948
C00651=1220.213,-47.164,-39.424,179.962,5.380,148.949
C00652=1220.218,-47.413,-39.413,179.960,5.380,148.950
C00653=1220.224,-47.663,-39.400,179.957,5.380,148.950
C00654=1220.228,-47.913,-39.387,179.955,5.380,148.951
C00655=1220.233,-48.163,-39.375,179.953,5.379,148.952
C00656=1220.239,-48.432,-39.362,179.950,5.379,148.953
C00657=1220.244,-48.702,-39.349,179.948,5.379,148.953
C00658=1220.250,-48.972,-39.335,179.945,5.379,148.954
C00659=1220.256,-49.242,-39.322,179.942,5.379,148.955
C00660=1220.261,-49.491,-39.309,179.940,5.378,148.955
C00661=1220.266,-49.742,-39.297,179.938,5.378,148.956
C00662=1220.271,-49.991,-39.285,179.935,5.378,148.957
C00663=1220.277,-50.241,-39.273,179.933,5.378,148.957
C00664=1220.281,-50.490,-39.261,179.930,5.378,148.958
C00665=1220.286,-50.739,-39.248,179.928,5.377,148.959
C00666=1220.291,-50.989,-39.236,179.926,5.378,148.960
C00667=1220.297,-51.239,-39.224,179.923,5.377,148.960
C00668=1220.302,-51.489,-39.212,179.921,5.377,148.961
C00669=1220.307,-51.738,-39.199,179.918,5.377,148.962
C00670=1220.313,-51.988,-39.187,179.915,5.376,148.962
C00671=1220.317,-52.238,-39.174,179.913,5.377,148.963
C00672=1220.323,-52.488,-39.162,179.911,5.376,148.964
C00673=1220.328,-52.737,-39.150,179.909,5.377,148.964
C00674=1220.332,-52.987,-39.138,179.906,5.376,148.965
C00675=1220.337,-53.236,-39.126,179.903,5.376,148.966
C00676=1220.343,-53.486,-39.114,179.901,5.376,148.967
C00677=1220.348,-53.735,-39.101,179.898,5.376,148.967
C00678=1220.353,-53.985,-39.089,179.896,5.376,148.968
C00679=1220.359,-54.235,-39.077,179.894,5.375,148.969
C00680=1220.363,-54.484,-39.066,179.891,5.375,148.969
C00681=1220.369,-54.734,-39.054,179.889,5.375,148.970
C00682=1220.374,-54.983,-39.041,179.886,5.375,148.971
C00683=1220.379,-55.233,-39.029,179.884,5.375,148.972
C00684=1220.384,-55.483,-39.017,179.882,5.375,148.972
C00685=1220.390,-55.733,-39.005,179.879,5.374,148.973
C00686=1220.394,-55.983,-38.993,179.877,5.375,148.974
C00687=1220.399,-56.232,-38.980,179.874,5.374,148.974
C00688=1220.404,-56.482,-38.969,179.873,5.374,148.975
C00689=1220.410,-56.731,-38.956,179.870,5.374,148.976
C00690=1220.415,-56.981,-38.944,179.868,5.374,148.976
C00691=1220.420,-57.231,-38.933,179.865,5.373,148.977
C00692=1220.425,-57.480,-38.920,179.862,5.373,148.978
C00693=1220.430,-57.730,-38.908,179.860,5.373,148.978
C00694=1220.436,-57.980,-38.896,179.858,5.373,148.979
C00695=1220.440,-58.229,-38.884,179.856,5.373,148.980
C00696=1220.446,-58.479,-38.873,179.853,5.373,148.980
C00697=1220.451,-58.729,-38.861,179.850,5.372,148.981
C00698=1220.456,-58.978,-38.848,179.848,5.373,148.982
C00699=1220.461,-59.228,-38.837,179.846,5.372,148.983
C00700=1220.466,-59.478,-38.825,179.843,5.373,148.983
C00701=1220.471,-59.727,-38.812,179.841,5.372,148.984
C00702=1220.477,-59.977,-38.800,179.839,5.372,148.985
C00703=1220.481,-60.227,-38.789,179.836,5.372,148.985
C00704=1220.487,-60.477,-38.777,179.833,5.371,148.986
C00705=1220.492,-60.726,-38.765,179.831,5.372,148.987
C00706=1220.497,-60.976,-38.753,179.829,5.371,148.987
C00707=1220.502,-61.226,-38.741,179.827,5.372,148.988
C00708=1220.508,-61.475,-38.730,179.824,5.371,148.989
C00709=1220.513,-61.724,-38.718,179.822,5.372,148.990
C00710=1220.518,-61.974,-38.706,179.819,5.371,148.990
C00711=1220.523,-62.224,-38.694,179.816,5.371,148.991
C00712=1220.529,-62.474,-38.682,179.815,5.371,148.991
C00713=1220.533,-62.723,-38.670,179.812,5.370,148.992
C00714=1220.539,-62.973,-38.658,179.810,5.370,148.993
C00715=1220.544,-63.223,-38.646,179.807,5.370,148.994
C00716=1220.549,-63.472,-38.635,179.805,5.370,148.994
C00717=1220.554,-63.722,-38.623,179.803,5.370,148.995
C00718=1220.559,-63.972,-38.612,179.800,5.369,148.996
C00719=1220.564,-64.221,-38.599,179.798,5.370,148.996
C00720=1220.569,-64.471,-38.588,179.795,5.369,148.997
C00721=1220.574,-64.721,-38.576,179.793,5.370,148.998
C00722=1220.580,-64.971,-38.564,179.790,5.369,148.999
C00723=1220.586,-65.220,-38.553,179.788,5.370,148.999
C00724=1220.590,-65.469,-38.542,179.786,5.369,149.000
C00725=1220.596,-65.719,-38.530,179.783,5.369,149.001
C00726=1220.600,-65.968,-38.518,179.781,5.369,149.001
C00727=1220.606,-66.218,-38.506,179.778,5.369,149.002
C00728=1220.611,-66.468,-38.494,179.776,5.369,149.003
C00729=1220.616,-66.718,-38.483,179.774,5.368,149.004
C00730=1220.621,-66.968,-38.471,179.771,5.369,149.004
C00731=1220.626,-67.217,-38.459,179.769,5.368,149.005
C00732=1220.632,-67.467,-38.448,179.766,5.368,149.006
C00733=1220.637,-67.717,-38.436,179.765,5.368,149.006
C00734=1220.642,-67.966,-38.425,179.762,5.367,149.007
C00735=1220.647,-68.216,-38.413,179.760,5.368,149.008
C00736=1220.652,-68.466,-38.402,179.757,5.367,149.008
C00737=1220.657,-68.716,-38.390,179.755,5.368,149.009
C00738=1220.662,-68.965,-38.378,179.752,5.367,149.010
C00739=1220.668,-69.215,-38.367,179.750,5.367,149.010
C00740=1220.673,-69.464,-38.356,179.748,5.367,149.011
C00741=1220.678,-69.714,-38.344,179.745,5.367,149.012
C00742=1220.684,-69.964,-38.332,179.743,5.367,149.012
C00743=1220.688,-70.214,-38.321,179.740,5.366,149.013
C00744=1220.694,-70.464,-38.309,179.738,5.367,149.014
C00745=1220.699,-70.713,-38.298,179.735,5.366,149.015
C00746=1220.705,-70.963,-38.286,179.733,5.367,149.015
C00747=1220.709,-71.212,-38.275,179.731,5.366,149.016
C00748=1220.715,-71.462,-38.263,179.729,5.367,149.017
C00749=1220.719,-71.712,-38.251,179.726,5.366,149.017
C00750=1220.725,-71.962,-38.239,179.724,5.366,149.018
C00751=1220.730,-72.211,-38.229,179.722,5.366,149.019
C00752=1220.736,-72.461,-38.217,179.719,5.365,149.019
C00753=1220.740,-72.710,-38.205,179.717,5.366,149.020
C00754=1220.746,-72.960,-38.193,179.714,5.365,149.021
C00755=1220.750,-73.210,-38.182,179.712,5.365,149.021
C00756=1220.756,-73.459,-38.171,179.709,5.365,149.022
C00757=1220.761,-73.709,-38.159,179.707,5.365,149.023
C00758=1220.766,-73.959,-38.149,179.705,5.365,149.024
C00759=1220.772,-74.209,-38.137,179.703,5.365,149.024
C00760=1220.777,-74.478,-38.124,179.700,5.365,149.025
C00761=1220.783,-74.749,-38.112,179.697,5.364,149.026
C00762=1220.788,-75.020,-38.100,179.695,5.365,149.026
C00763=1220.794,-75.290,-38.088,179.692,5.365,149.027
C00764=1220.799,-75.540,-38.076,179.689,5.364,149.028
C00765=1220.804,-75.790,-38.065,179.687,5.365,149.029
C00766=1220.810,-76.040,-38.053,179.685,5.364,149.029
C00767=1220.815,-76.289,-38.043,179.683,5.364,149.030
C00768=1220.820,-76.538,-38.031,179.680,5.364,149.031
C00769=1220.825,-76.788,-38.019,179.678,5.364,149.031
C00770=1220.831,-77.038,-38.009,179.676,5.364,149.032
C00771=1220.836,-77.288,-37.997,179.673,5.364,149.033
C00772=1220.841,-77.537,-37.986,179.671,5.363,149.033
C00773=1220.845,-77.787,-37.975,179.669,5.364,149.034
C00774=1220.852,-78.036,-37.963,179.666,5.363,149.035
C00775=1220.857,-78.287,-37.953,179.664,5.364,149.036
C00776=1220.861,-78.536,-37.941,179.661,5.363,149.036
C00777=1220.867,-78.786,-37.929,179.659,5.363,149.037
C00778=1220.872,-79.035,-37.919,179.656,5.363,149.038
C00779=1220.877,-79.285,-37.908,179.654,5.363,149.038
C00780=1220.882,-79.535,-37.896,179.652,5.363,149.039
C00781=1220.888,-79.784,-37.885,179.650,5.362,149.040
C00782=1220.892,-80.034,-37.874,179.647,5.363,149.040
C00783=1220.898,-80.284,-37.863,179.645,5.362,149.041
C00784=1220.903,-80.534,-37.851,179.643,5.362,149.042
C00785=1220.908,-80.783,-37.840,179.640,5.362,149.042
C00786=1220.914,-81.033,-37.829,179.638,5.362,149.043
C00787=1220.918,-81.283,-37.818,179.635,5.362,149.044
C00788=1220.924,-81.532,-37.807,179.633,5.362,149.045
C00789=1220.929,-81.782,-37.796,179.630,5.362,149.045
C00790=1220.934,-82.032,-37.785,179.628,5.362,149.046
C00791=1220.940,-82.281,-37.774,179.626,5.362,149.047
C00792=1220.945,-82.531,-37.763,179.624,5.362,149.047
C00793=1220.950,-82.781,-37.751,179.621,5.361,149.048
C00794=1220.955,-83.030,-37.740,179.619,5.361,149.049
C00795=1220.960,-83.280,-37.730,179.617,5.361,149.049
C00796=1220.965,-83.530,-37.718,179.614,5.361,149.050
C00797=1220.971,-83.780,-37.708,179.612,5.361,149.051
C00798=1220.976,-84.030,-37.696,179.609,5.361,149.051
C00799=1220.981,-84.279,-37.685,179.607,5.361,149.052
C00800=1220.986,-84.529,-37.675,179.605,5.361,149.053
C00801=1220.991,-84.778,-37.664,179.602,5.361,149.054
C00802=1220.997,-85.029,-37.652,179.600,5.360,149.054
C00803=1221.002,-85.278,-37.641,179.598,5.361,149.055
C00804=1221.007,-85.527,-37.630,179.595,5.360,149.056
C00805=1221.012,-85.778,-37.620,179.593,5.360,149.056
C00806=1221.018,-86.027,-37.608,179.591,5.360,149.057
C00807=1221.023,-86.277,-37.597,179.589,5.360,149.058
C00808=1221.028,-86.526,-37.587,179.586,5.360,149.058
C00809=1221.033,-86.776,-37.576,179.584,5.360,149.059
C00810=1221.038,-87.026,-37.565,179.581,5.360,149.060
C00811=1221.043,-87.275,-37.554,179.579,5.360,149.060
C00812=1221.049,-87.525,-37.543,179.576,5.360,149.061
C00813=1221.054,-87.776,-37.532,179.574,5.360,149.062
C00814=1221.059,-88.025,-37.521,179.572,5.360,149.063
C00815=1221.064,-88.275,-37.511,179.570,5.360,149.063
C00816=1221.069,-88.524,-37.500,179.567,5.359,149.064
C00817=1221.074,-88.774,-37.489,179.565,5.360,149.065
C00818=1221.080,-89.024,-37.477,179.563,5.359,149.065
C00819=1221.085,-89.274,-37.467,179.561,5.359,149.066
C00820=1221.090,-89.523,-37.456,179.558,5.359,149.067
C00821=1221.096,-89.773,-37.445,179.556,5.359,149.067
C00822=1221.100,-90.022,-37.434,179.553,5.359,149.068
C00823=1221.106,-90.272,-37.424,179.551,5.359,149.069
C00824=1221.111,-90.522,-37.413,179.548,5.359,149.069
C00825=1221.116,-90.772,-37.402,179.546,5.359,149.070
C00826=1221.121,-91.021,-37.392,179.544,5.358,149.071
C00827=1221.127,-91.271,-37.380,179.542,5.359,149.071
C00828=1221.132,-91.521,-37.370,179.539,5.358,149.072
C00829=1221.137,-91.771,-37.359,179.537,5.359,149.073
C00830=1221.142,-92.020,-37.348,179.535,5.358,149.074
C00831=1221.147,-92.270,-37.338,179.532,5.359,149.074
C00832=1221.153,-92.519,-37.327,179.530,5.358,149.075
C00833=1221.158,-92.769,-37.316,179.528,5.359,149.076
C00834=1221.163,-93.019,-37.306,179.525,5.358,149.076
C00835=1221.168,-93.268,-37.295,179.523,5.358,149.077
C00836=1221.173,-93.519,-37.284,179.521,5.358,149.078
C00837=1221.179,-93.768,-37.274,179.519,5.358,149.078
C00838=1221.183,-94.018,-37.263,179.516,5.358,149.079
C00839=1221.189,-94.267,-37.252,179.514,5.358,149.080
C00840=1221.194,-94.518,-37.242,179.511,5.357,149.080
C00841=1221.199,-94.767,-37.231,179.509,5.358,149.081
C00842=1221.205,-95.017,-37.220,179.506,5.357,149.082
C00843=1221.211,-95.267,-37.210,179.504,5.358,149.083
C00844=1221.215,-95.516,-37.198,179.502,5.357,149.083
C00845=1221.221,-95.766,-37.188,179.500,5.357,149.084
C00846=1221.226,-96.016,-37.177,179.497,5.357,149.084
C00847=1221.231,-96.266,-37.167,179.495,5.357,149.085
C00848=1221.236,-96.515,-37.156,179.493,5.357,149.086
C00849=1221.242,-96.765,-37.146,179.491,5.357,149.087
C00850=1221.247,-97.015,-37.135,179.488,5.357,149.087
C00851=1221.252,-97.265,-37.125,179.486,5.357,149.088
C00852=1221.258,-97.514,-37.114,179.483,5.357,149.089
C00853=1221.263,-97.764,-37.103,179.481,5.357,149.089
C00854=1221.267,-98.013,-37.094,179.479,5.356,149.090
C00855=1221.272,-98.263,-37.083,179.477,5.357,149.091
C00856=1221.278,-98.513,-37.073,179.474,5.356,149.091
C00857=1221.283,-98.762,-37.062,179.472,5.357,149.092
C00858=1221.288,-99.012,-37.052,179.469,5.356,149.093
C00859=1221.293,-99.262,-37.041,179.467,5.356,149.093
C00860=1221.299,-99.512,-37.031,179.465,5.356,149.094
C00861=1221.304,-99.762,-37.020,179.462,5.356,149.095
C00862=1221.309,-100.011,-37.009,179.460,5.356,149.095
C00863=1221.315,-100.260,-36.999,179.458,5.356,149.096
C00864=1221.320,-100.532,-36.988,179.455,5.356,149.097
C00865=1221.326,-100.803,-36.977,179.452,5.355,149.098
C00866=1221.331,-101.075,-36.966,179.450,5.356,149.098
C00867=1221.337,-101.345,-36.954,179.448,5.355,149.099
C00868=1221.342,-101.595,-36.943,179.445,5.356,149.100
C00869=1221.348,-101.845,-36.933,179.443,5.355,149.101
C00870=1221.353,-102.095,-36.922,179.441,5.355,149.101
C00871=1221.358,-102.344,-36.913,179.438,5.355,149.102
C00872=1221.363,-102.594,-36.903,179.436,5.355,149.103
C00873=1221.368,-102.844,-36.892,179.434,5.355,149.103
C00874=1221.374,-103.094,-36.882,179.432,5.355,149.104
C00875=1221.379,-103.343,-36.871,179.429,5.355,149.105
C00876=1221.384,-103.593,-36.860,179.427,5.355,149.105
C00877=1221.390,-103.842,-36.850,179.425,5.354,149.106
C00878=1221.394,-104.092,-36.840,179.423,5.355,149.107
C00879=1221.400,-104.342,-36.830,179.420,5.354,149.107
C00880=1221.405,-104.592,-36.819,179.418,5.355,149.108
C00881=1221.410,-104.842,-36.809,179.415,5.354,149.109
C00882=1221.416,-105.091,-36.799,179.413,5.355,149.109
C00883=1221.421,-105.341,-36.788,179.410,5.354,149.110
C00884=1221.426,-105.591,-36.779,179.409,5.354,149.111
C00885=1221.431,-105.840,-36.769,179.407,5.355,149.111
C00886=1221.436,-106.090,-36.758,179.404,5.354,149.112
C00887=1221.442,-106.340,-36.748,179.402,5.355,149.113
C00888=1221.447,-106.590,-36.737,179.399,5.354,149.114
C00889=1221.452,-106.839,-36.728,179.397,5.354,149.114
C00890=1221.457,-107.089,-36.717,179.394,5.354,149.115
C00891=1221.462,-107.339,-36.707,179.393,5.354,149.115
C00892=1221.468,-107.589,-36.697,179.390,5.354,149.116
C00893=1221.474,-107.838,-36.686,179.388,5.354,149.117
C00894=1221.478,-108.088,-36.676,179.385,5.354,149.118
C00895=1221.484,-108.338,-36.666,179.383,5.354,149.118
C00896=1221.489,-108.587,-36.656,179.381,5.353,149.119
C00897=1221.494,-108.837,-36.645,179.379,5.354,149.120
C00898=1221.499,-109.087,-36.637,179.376,5.353,149.120
C00899=1221.505,-109.337,-36.626,179.374,5.353,149.121
C00900=1221.510,-109.587,-36.616,179.372,5.353,149.122
C00901=1221.515,-109.837,-36.606,179.370,5.353,149.122
C00902=1221.520,-110.086,-36.596,179.367,5.353,149.123
C00903=1221.526,-110.335,-36.586,179.365,5.353,149.124
C00904=1221.531,-110.586,-36.575,179.363,5.353,149.124
C00905=1221.537,-110.835,-36.565,179.360,5.353,149.125
C00906=1221.541,-111.084,-36.555,179.358,5.353,149.126
C00907=1221.547,-111.335,-36.545,179.356,5.353,149.126
C00908=1221.552,-111.585,-36.535,179.354,5.353,149.127
C00909=1221.557,-111.834,-36.526,179.351,5.353,149.128
C00910=1221.563,-112.084,-36.515,179.349,5.353,149.128
C00911=1221.568,-112.334,-36.505,179.347,5.352,149.129
C00912=1221.573,-112.583,-36.495,179.345,5.353,149.130
C00913=1221.578,-112.833,-36.485,179.342,5.352,149.130
C00914=1221.584,-113.084,-36.475,179.340,5.353,149.131
C00915=1221.588,-113.333,-36.466,179.337,5.352,149.132
C00916=1221.594,-113.582,-36.455,179.336,5.352,149.132
C00917=1221.600,-113.832,-36.445,179.333,5.352,149.133
C00918=1221.604,-114.082,-36.435,179.331,5.352,149.134
C00919=1221.610,-114.332,-36.426,179.328,5.352,149.135
C00920=1221.615,-114.582,-36.415,179.326,5.352,149.135
C00921=1221.620,-114.831,-36.406,179.324,5.353,149.136
C00922=1221.625,-115.081,-36.395,179.322,5.352,149.136
C00923=1221.631,-115.331,-36.386,179.320,5.352,149.137
C00924=1221.636,-115.580,-36.376,179.317,5.352,149.138
C00925=1221.642,-115.830,-36.366,179.315,5.352,149.139
C00926=1221.647,-116.080,-36.355,179.312,5.352,149.139
C00927=1221.652,-116.330,-36.346,179.310,5.352,149.140
C00928=1221.657,-116.580,-36.336,179.308,5.351,149.140
C00929=1221.662,-116.829,-36.327,179.306,5.352,149.141
C00930=1221.668,-117.079,-36.317,179.303,5.351,149.142
C00931=1221.673,-117.329,-36.307,179.301,5.352,149.143
C00932=1221.678,-117.578,-36.297,179.298,5.351,149.143
C00933=1221.684,-117.828,-36.287,179.297,5.351,149.144
C00934=1221.689,-118.078,-36.278,179.295,5.352,149.145
C00935=1221.694,-118.327,-36.268,179.292,5.351,149.145
C00936=1221.699,-118.577,-36.258,179.290,5.352,149.146
C00937=1221.704,-118.827,-36.248,179.287,5.351,149.147
C00938=1221.710,-119.077,-36.238,179.286,5.351,149.147
C00939=1221.715,-119.326,-36.228,179.283,5.351,149.148
C00940=1221.721,-119.576,-36.219,179.281,5.351,149.149
C00941=1221.725,-119.826,-36.209,179.278,5.351,149.149
C00942=1221.731,-120.076,-36.199,179.276,5.351,149.150
C00943=1221.736,-120.326,-36.190,179.273,5.351,149.151
C00944=1221.741,-120.575,-36.180,179.272,5.351,149.151
C00945=1221.747,-120.825,-36.171,179.270,5.351,149.152
C00946=1221.752,-121.075,-36.160,179.267,5.351,149.153
C00947=1221.756,-121.325,-36.150,179.265,5.351,149.153
C00948=1221.762,-121.575,-36.141,179.262,5.351,149.154
C00949=1221.767,-121.824,-36.131,179.261,5.351,149.155
C00950=1221.773,-122.074,-36.122,179.258,5.350,149.155
C00951=1221.778,-122.323,-36.112,179.256,5.351,149.156
C00952=1221.784,-122.574,-36.103,179.253,5.350,149.157
C00953=1221.788,-122.823,-36.093,179.252,5.350,149.157
C00954=1221.794,-123.073,-36.083,179.249,5.350,149.158
C00955=1221.799,-123.323,-36.074,179.247,5.350,149.159
C00956=1221.805,-123.572,-36.063,179.245,5.350,149.159
C00957=1221.810,-123.822,-36.055,179.242,5.350,149.160
C00958=1221.815,-124.072,-36.044,179.240,5.350,149.161
C00959=1221.820,-124.322,-36.035,179.238,5.350,149.161
C00960=1221.825,-124.572,-36.025,179.236,5.350,149.162
C00961=1221.831,-124.822,-36.016,179.233,5.350,149.163
C00962=1221.835,-125.071,-36.006,179.231,5.350,149.163
C00963=1221.841,-125.321,-35.997,179.229,5.349,149.164
C00964=1221.846,-125.570,-35.987,179.227,5.350,149.165
C00965=1221.852,-125.821,-35.978,179.224,5.350,149.165
C00966=1221.857,-126.070,-35.968,179.222,5.350,149.166
C00967=1221.863,-126.320,-35.959,179.220,5.350,149.167
C00968=1221.441,-126.331,-35.995,179.216,5.353,149.169
C00969=1221.435,-126.081,-36.005,179.218,5.353,149.168
C00970=1221.430,-125.831,-36.014,179.220,5.352,149.167
C00971=1221.424,-125.581,-36.024,179.222,5.353,149.167
C00972=1221.420,-125.332,-36.033,179.224,5.353,149.166
C00973=1221.414,-125.082,-36.042,179.227,5.353,149.165
C00974=1221.409,-124.833,-36.052,179.229,5.353,149.165
C00975=1221.404,-124.582,-36.062,179.231,5.354,149.164
C00976=1221.399,-124.332,-36.072,179.233,5.353,149.163
C00977=1221.394,-124.083,-36.081,179.236,5.354,149.163
C00978=1221.388,-123.833,-36.091,179.238,5.353,149.162
C00979=1221.383,-123.583,-36.100,179.241,5.354,149.161
C00980=1221.377,-123.334,-36.110,179.242,5.354,149.161
C00981=1221.372,-123.084,-36.119,179.244,5.353,149.160
C00982=1221.366,-122.834,-36.129,179.247,5.354,149.159
C00983=1221.362,-122.584,-36.139,179.249,5.353,149.159
C00984=1221.356,-122.334,-36.149,179.252,5.354,149.158
C00985=1221.351,-122.085,-36.158,179.253,5.354,149.157
C00986=1221.345,-121.835,-36.168,179.256,5.354,149.157
C00987=1221.341,-121.586,-36.177,179.258,5.354,149.156
C00988=1221.335,-121.335,-36.187,179.261,5.354,149.155
C00989=1221.330,-121.085,-36.197,179.263,5.354,149.155
C00990=1221.325,-120.836,-36.207,179.265,5.355,149.154
C00991=1221.320,-120.586,-36.216,179.267,5.354,149.153
C00992=1221.314,-120.336,-36.226,179.269,5.354,149.153
C00993=1221.309,-120.087,-36.235,179.272,5.354,149.152
C00994=1221.303,-119.837,-36.245,179.274,5.354,149.151
C00995=1221.299,-119.587,-36.255,179.276,5.355,149.151
C00996=1221.293,-119.337,-36.265,179.278,5.354,149.150
C00997=1221.288,-119.088,-36.274,179.281,5.355,149.149
C00998=1221.283,-118.838,-36.285,179.283,5.354,149.149
C00999=1221.278,-118.588,-36.293,179.286,5.355,149.148
C01000=1221.273,-118.338,-36.304,179.287,5.355,149.147
C01001=1221.267,-118.089,-36.314,179.290,5.355,149.147
C01002=1221.262,-117.839,-36.323,179.292,5.355,149.146
C01003=1221.256,-117.589,-36.333,179.294,5.354,149.145
C01004=1221.251,-117.340,-36.343,179.297,5.355,149.145
C01005=1221.246,-117.089,-36.353,179.299,5.355,149.144
C01006=1221.241,-116.840,-36.362,179.301,5.355,149.143
C01007=1221.236,-116.590,-36.373,179.303,5.355,149.143
C01008=1221.230,-116.341,-36.383,179.306,5.355,149.142
C01009=1221.225,-116.091,-36.392,179.308,5.355,149.141
C01010=1221.220,-115.841,-36.402,179.310,5.356,149.141
C01011=1221.215,-115.591,-36.412,179.312,5.355,149.140
C01012=1221.209,-115.341,-36.421,179.315,5.356,149.139
C01013=1221.203,-115.092,-36.432,179.317,5.355,149.139
C01014=1221.199,-114.842,-36.442,179.320,5.356,149.138
C01015=1221.194,-114.592,-36.452,179.322,5.355,149.137
C01016=1221.188,-114.343,-36.462,179.324,5.355,149.137
C01017=1221.183,-114.093,-36.471,179.326,5.356,149.136
C01018=1221.178,-113.843,-36.481,179.328,5.355,149.135
C01019=1221.172,-113.593,-36.492,179.331,5.356,149.134
C01020=1221.167,-113.344,-36.501,179.333,5.355,149.134
C01021=1221.161,-113.094,-36.511,179.336,5.356,149.133
C01022=1221.156,-112.843,-36.521,179.337,5.356,149.133
C01023=1221.152,-112.594,-36.531,179.340,5.356,149.132
C01024=1221.146,-112.345,-36.541,179.342,5.356,149.131
C01025=1221.140,-112.095,-36.551,179.345,5.356,149.130
C01026=1221.136,-111.845,-36.561,179.347,5.356,149.130
C01027=1221.130,-111.595,-36.571,179.349,5.357,149.129
C01028=1221.125,-111.345,-36.581,179.351,5.356,149.128
C01029=1221.120,-111.096,-36.591,179.354,5.357,149.128
C01030=1221.115,-110.846,-36.601,179.356,5.356,149.127
C01031=1221.109,-110.596,-36.611,179.358,5.356,149.126
C01032=1221.104,-110.347,-36.622,179.361,5.356,149.126
C01033=1221.099,-110.097,-36.632,179.363,5.356,149.125
C01034=1221.093,-109.847,-36.641,179.365,5.357,149.124
C01035=1221.088,-109.597,-36.651,179.367,5.357,149.124
C01036=1221.083,-109.347,-36.662,179.370,5.357,149.123
C01037=1221.078,-109.098,-36.672,179.372,5.357,149.122
C01038=1221.072,-108.848,-36.682,179.375,5.357,149.122
C01039=1221.067,-108.598,-36.692,179.377,5.357,149.121
C01040=1221.062,-108.348,-36.703,179.379,5.357,149.120
C01041=1221.057,-108.099,-36.712,179.381,5.357,149.120
C01042=1221.052,-107.849,-36.723,179.384,5.357,149.119
C01043=1221.046,-107.599,-36.733,179.386,5.357,149.118
C01044=1221.041,-107.350,-36.743,179.388,5.358,149.118
C01045=1221.036,-107.100,-36.753,179.391,5.357,149.117
C01046=1221.031,-106.850,-36.763,179.393,5.358,149.116
C01047=1221.025,-106.601,-36.774,179.395,5.358,149.116
C01048=1221.020,-106.351,-36.784,179.397,5.358,149.115
C01049=1221.015,-106.101,-36.794,179.400,5.358,149.114
C01050=1221.010,-105.852,-36.804,179.402,5.358,149.113
C01051=1221.005,-105.602,-36.815,179.404,5.358,149.113
C01052=1220.999,-105.352,-36.825,179.406,5.357,149.112
C01053=1220.994,-105.102,-36.835,179.409,5.358,149.112
C01054=1220.989,-104.852,-36.846,179.411,5.358,149.111
C01055=1220.984,-104.603,-36.855,179.413,5.358,149.110
C01056=1220.979,-104.353,-36.866,179.415,5.358,149.109
C01057=1220.973,-104.103,-36.876,179.418,5.358,149.109
C01058=1220.968,-103.854,-36.886,179.420,5.358,149.108
C01059=1220.963,-103.603,-36.897,179.423,5.358,149.107
C01060=1220.957,-103.354,-36.907,179.424,5.358,149.107
C01061=1220.953,-103.104,-36.917,179.427,5.359,149.106
C01062=1220.947,-102.854,-36.927,179.429,5.358,149.105
C01063=1220.941,-102.605,-36.937,179.432,5.359,149.105
C01064=1220.936,-102.355,-36.948,179.434,5.358,149.104
C01065=1220.931,-102.105,-36.958,179.437,5.359,149.103
C01066=1220.926,-101.855,-36.969,179.439,5.358,149.103
C01067=1220.921,-101.606,-36.980,179.441,5.359,149.102
C01068=1220.916,-101.356,-36.990,179.443,5.359,149.101
C01069=1220.910,-101.085,-37.001,179.446,5.359,149.101
C01070=1220.904,-100.813,-37.012,179.448,5.359,149.100
C01071=1220.899,-100.542,-37.023,179.451,5.359,149.099
C01072=1220.892,-100.272,-37.035,179.454,5.359,149.098
C01073=1220.888,-100.022,-37.045,179.456,5.359,149.098
C01074=1220.883,-99.772,-37.055,179.458,5.360,149.097
C01075=1220.878,-99.522,-37.066,179.460,5.360,149.096
C01076=1220.872,-99.273,-37.076,179.463,5.360,149.096
C01077=1220.867,-99.023,-37.087,179.465,5.360,149.095
C01078=1220.862,-98.773,-37.098,179.468,5.360,149.094
C01079=1220.856,-98.524,-37.108,179.470,5.360,149.093
C01080=1220.851,-98.274,-37.118,179.472,5.360,149.093
C01081=1220.846,-98.024,-37.129,179.474,5.360,149.092
C01082=1220.841,-97.775,-37.140,179.477,5.360,149.091
C01083=1220.835,-97.525,-37.150,179.479,5.360,149.091
C01084=1220.830,-97.275,-37.161,179.481,5.361,149.090
C01085=1220.825,-97.025,-37.171,179.483,5.360,149.089
C01086=1220.820,-96.775,-37.181,179.486,5.361,149.089
C01087=1220.814,-96.526,-37.192,179.488,5.360,149.088
C01088=1220.809,-96.276,-37.203,179.491,5.361,149.087
C01089=1220.804,-96.026,-37.213,179.493,5.360,149.087
C01090=1220.799,-95.776,-37.224,179.496,5.361,149.086
C01091=1220.793,-95.527,-37.235,179.497,5.361,149.085
C01092=1220.788,-95.277,-37.245,179.500,5.361,149.085
C01093=1220.783,-95.027,-37.255,179.502,5.361,149.084
C01094=1220.778,-94.778,-37.267,179.505,5.361,149.083
C01095=1220.773,-94.528,-37.277,179.507,5.361,149.083
C01096=1220.768,-94.278,-37.287,179.509,5.361,149.082
C01097=1220.762,-94.029,-37.298,179.512,5.361,149.081
C01098=1220.757,-93.779,-37.309,179.514,5.361,149.080
C01099=1220.752,-93.529,-37.319,179.516,5.361,149.080
C01100=1220.747,-93.280,-37.330,179.518,5.362,149.079
C01101=1220.741,-93.030,-37.341,179.521,5.362,149.078
C01102=1220.736,-92.780,-37.351,179.523,5.362,149.078
C01103=1220.731,-92.531,-37.362,179.525,5.362,149.077
C01104=1220.726,-92.281,-37.373,179.528,5.362,149.076
C01105=1220.721,-92.031,-37.383,179.530,5.362,149.076
C01106=1220.715,-91.781,-37.395,179.533,5.362,149.075
C01107=1220.710,-91.532,-37.405,179.535,5.362,149.074
C01108=1220.705,-91.282,-37.416,179.538,5.362,149.073
C01109=1220.700,-91.032,-37.427,179.540,5.362,149.073
C01110=1220.694,-90.782,-37.437,179.542,5.363,149.072
C01111=1220.690,-90.533,-37.448,179.544,5.362,149.072
C01112=1220.684,-90.283,-37.459,179.547,5.363,149.071
C01113=1220.679,-90.033,-37.470,179.549,5.362,149.070
C01114=1220.674,-89.784,-37.480,179.551,5.363,149.069
C01115=1220.669,-89.534,-37.491,179.553,5.362,149.069
C01116=1220.663,-89.284,-37.503,179.556,5.363,149.068
C01117=1220.658,-89.034,-37.513,179.558,5.363,149.067
C01118=1220.653,-88.784,-37.524,179.561,5.363,149.067
C01119=1220.647,-88.535,-37.534,179.563,5.363,149.066
C01120=1220.643,-88.285,-37.546,179.565,5.363,149.065
C01121=1220.637,-88.036,-37.556,179.567,5.363,149.065
C01122=1220.632,-87.786,-37.567,179.570,5.364,149.064
C01123=1220.627,-87.536,-37.578,179.572,5.363,149.063
C01124=1220.621,-87.287,-37.589,179.575,5.364,149.063
C01125=1220.616,-87.036,-37.600,179.577,5.363,149.062
C01126=1220.612,-86.787,-37.611,179.579,5.364,149.061
C01127=1220.606,-86.537,-37.621,179.581,5.363,149.060
C01128=1220.601,-86.287,-37.633,179.584,5.364,149.060
C01129=1220.595,-86.038,-37.643,179.586,5.363,149.059
C01130=1220.590,-85.788,-37.655,179.588,5.364,149.059
C01131=1220.585,-85.538,-37.665,179.591,5.364,149.058
C01132=1220.580,-85.289,-37.676,179.593,5.364,149.057
C01133=1220.575,-85.039,-37.688,179.595,5.364,149.056
C01134=1220.570,-84.789,-37.699,179.598,5.364,149.056
C01135=1220.564,-84.540,-37.710,179.600,5.364,149.055
C01136=1220.559,-84.290,-37.720,179.603,5.364,149.054
C01137=1220.554,-84.041,-37.731,179.605,5.364,149.054
C01138=1220.549,-83.791,-37.743,179.607,5.365,149.053
C01139=1220.544,-83.540,-37.753,179.610,5.365,149.052
C01140=1220.538,-83.292,-37.764,179.612,5.365,149.051
C01141=1220.533,-83.041,-37.775,179.615,5.365,149.051
C01142=1220.528,-82.791,-37.787,179.617,5.365,149.050
C01143=1220.523,-82.542,-37.798,179.619,5.366,149.050
C01144=1220.518,-82.292,-37.808,179.621,5.365,149.049
C01145=1220.513,-82.043,-37.820,179.624,5.366,149.048
C01146=1220.507,-81.793,-37.831,179.626,5.365,149.047
C01147=1220.502,-81.543,-37.842,179.629,5.366,149.047
C01148=1220.497,-81.293,-37.853,179.631,5.365,149.046
C01149=1220.492,-81.044,-37.865,179.633,5.366,149.045
C01150=1220.486,-80.794,-37.875,179.636,5.365,149.045
C01151=1220.481,-80.544,-37.886,179.638,5.366,149.044
C01152=1220.477,-80.295,-37.898,179.640,5.366,149.043
C01153=1220.470,-80.045,-37.909,179.643,5.366,149.042
C01154=1220.466,-79.795,-37.920,179.645,5.366,149.042
C01155=1220.461,-79.546,-37.931,179.647,5.367,149.041
C01156=1220.455,-79.296,-37.942,179.649,5.366,149.041
C01157=1220.450,-79.046,-37.953,179.652,5.367,149.040
C01158=1220.445,-78.797,-37.964,179.655,5.367,149.039
C01159=1220.440,-78.547,-37.976,179.657,5.367,149.038
C01160=1220.434,-78.297,-37.987,179.659,5.367,149.038
C01161=1220.430,-78.047,-37.998,179.662,5.367,149.037
C01162=1220.424,-77.798,-38.010,179.664,5.367,149.036
C01163=1220.419,-77.548,-38.021,179.666,5.367,149.036
C01164=1220.413,-77.299,-38.033,179.669,5.367,149.035
C01165=1220.408,-77.048,-38.043,179.671,5.367,149.034
C01166=1220.404,-76.799,-38.054,179.674,5.367,149.033
C01167=1220.398,-76.550,-38.066,179.676,5.367,149.033
C01168=1220.393,-76.300,-38.077,179.678,5.368,149.032
C01169=1220.388,-76.050,-38.089,179.680,5.368,149.032
C01170=1220.383,-75.800,-38.100,179.683,5.368,149.031
C01171=1220.377,-75.551,-38.111,179.685,5.368,149.030
C01172=1220.372,-75.301,-38.122,179.688,5.368,149.029
C01173=1220.366,-75.030,-38.135,179.690,5.369,149.029
C01174=1220.361,-74.761,-38.147,179.693,5.368,149.028
C01175=1220.355,-74.490,-38.159,179.695,5.368,149.027
C01176=1220.350,-74.219,-38.171,179.698,5.369,149.026
C01177=1220.344,-73.969,-38.183,179.700,5.368,149.026
C01178=1220.339,-73.720,-38.194,179.703,5.369,149.025
C01179=1220.334,-73.470,-38.206,179.705,5.368,149.024
C01180=1220.329,-73.220,-38.217,179.708,5.369,149.024
C01181=1220.324,-72.971,-38.229,179.710,5.369,149.023
C01182=1220.318,-72.721,-38.240,179.712,5.369,149.022
C01183=1220.314,-72.472,-38.251,179.715,5.370,149.022
C01184=1220.308,-72.222,-38.263,179.717,5.370,149.021
C01185=1220.303,-71.972,-38.275,179.719,5.370,149.020
C01186=1220.298,-71.722,-38.286,179.721,5.370,149.020
C01187=1220.292,-71.473,-38.297,179.724,5.370,149.019
C01188=1220.287,-71.223,-38.308,179.726,5.370,149.018
C01189=1220.282,-70.973,-38.320,179.729,5.370,149.017
C01190=1220.277,-70.723,-38.332,179.731,5.370,149.017
C01191=1220.272,-70.474,-38.343,179.734,5.370,149.016
C01192=1220.267,-70.224,-38.355,179.736,5.371,149.015
C01193=1220.261,-69.975,-38.366,179.738,5.370,149.015
C01194=1220.256,-69.725,-38.378,179.741,5.371,149.014
C01195=1220.251,-69.475,-38.389,179.743,5.370,149.013
C01196=1220.246,-69.225,-38.401,179.746,5.371,149.012
C01197=1220.241,-68.975,-38.413,179.748,5.371,149.012
C01198=1220.236,-68.726,-38.424,179.751,5.371,149.011
C01199=1220.230,-68.476,-38.436,179.752,5.371,149.011
C01200=1220.225,-68.227,-38.447,179.755,5.372,149.010
C01201=1220.220,-67.977,-38.459,179.757,5.372,149.009
C01202=1220.215,-67.727,-38.470,179.760,5.372,149.008
C01203=1220.210,-67.477,-38.482,179.762,5.372,149.008
C01204=1220.205,-67.228,-38.493,179.764,5.372,149.007
C01205=1220.200,-66.978,-38.506,179.767,5.372,149.006
C01206=1220.194,-66.728,-38.518,179.769,5.372,149.006
C01207=1220.189,-66.479,-38.529,179.772,5.372,149.005
C01208=1220.184,-66.230,-38.540,179.774,5.372,149.004
C01209=1220.179,-65.980,-38.552,179.777,5.372,149.003
C01210=1220.173,-65.730,-38.564,179.779,5.373,149.003
C01211=1220.168,-65.480,-38.576,179.781,5.373,149.002
C01212=1220.163,-65.230,-38.587,179.784,5.373,149.001
C01213=1220.158,-64.980,-38.599,179.786,5.373,149.001
C01214=1220.154,-64.731,-38.611,179.789,5.373,149.000
C01215=1220.148,-64.481,-38.623,179.791,5.373,148.999
C01216=1220.143,-64.232,-38.634,179.793,5.373,148.999
C01217=1220.137,-63.983,-38.645,179.796,5.374,148.998
C01218=1220.132,-63.733,-38.657,179.798,5.374,148.997
C01219=1220.127,-63.483,-38.669,179.800,5.374,148.997
C01220=1220.122,-63.233,-38.680,179.802,5.374,148.996
C01221=1220.117,-62.984,-38.693,179.805,5.374,148.995
C01222=1220.111,-62.734,-38.705,179.807,5.374,148.995
C01223=1220.107,-62.484,-38.716,179.810,5.374,148.994
C01224=1220.101,-62.234,-38.728,179.813,5.375,148.993
C01225=1220.096,-61.984,-38.740,179.815,5.375,148.992
C01226=1220.091,-61.735,-38.752,179.817,5.375,148.992
C01227=1220.086,-61.485,-38.764,179.819,5.375,148.991
C01228=1220.080,-61.235,-38.776,179.822,5.375,148.990
C01229=1220.076,-60.986,-38.787,179.824,5.375,148.990
C01230=1220.071,-60.737,-38.800,179.827,5.375,148.989
C01231=1220.065,-60.487,-38.812,179.829,5.376,148.988
C01232=1220.060,-60.237,-38.823,179.832,5.375,148.987
C01233=1220.055,-59.987,-38.835,179.834,5.376,148.987
C01234=1220.050,-59.738,-38.847,179.836,5.375,148.986
C01235=1220.045,-59.488,-38.859,179.839,5.376,148.985
C01236=1220.040,-59.238,-38.871,179.841,5.376,148.985
C01237=1220.035,-58.989,-38.883,179.844,5.376,148.984
C01238=1220.029,-58.739,-38.895,179.846,5.377,148.983
C01239=1220.024,-58.489,-38.907,179.848,5.377,148.983
C01240=1220.019,-58.240,-38.919,179.851,5.377,148.982
C01241=1220.014,-57.990,-38.931,179.853,5.377,148.981
C01242=1220.009,-57.740,-38.943,179.855,5.377,148.981
C01243=1220.004,-57.491,-38.955,179.858,5.378,148.980
C01244=1219.999,-57.241,-38.967,179.860,5.377,148.979
C01245=1219.993,-56.991,-38.978,179.863,5.378,148.979
C01246=1219.988,-56.742,-38.991,179.865,5.377,148.978
C01247=1219.983,-56.492,-39.003,179.868,5.378,148.977
C01248=1219.977,-56.242,-39.015,179.870,5.378,148.976
C01249=1219.973,-55.993,-39.027,179.872,5.378,148.976
C01250=1219.968,-55.743,-39.039,179.875,5.378,148.975
C01251=1219.962,-55.494,-39.051,179.877,5.378,148.974
C01252=1219.957,-55.244,-39.063,179.880,5.379,148.974
C01253=1219.952,-54.994,-39.075,179.882,5.378,148.973
C01254=1219.947,-54.745,-39.087,179.885,5.379,148.972
C01255=1219.942,-54.495,-39.099,179.887,5.379,148.972
C01256=1219.937,-54.246,-39.112,179.889,5.379,148.971
C01257=1219.931,-53.996,-39.123,179.892,5.379,148.970
C01258=1219.926,-53.746,-39.136,179.894,5.379,148.969
C01259=1219.921,-53.496,-39.148,179.897,5.379,148.969
C01260=1219.916,-53.247,-39.159,179.899,5.380,148.968
C01261=1219.911,-52.998,-39.172,179.901,5.380,148.967
C01262=1219.905,-52.748,-39.184,179.904,5.380,148.967
C01263=1219.901,-52.498,-39.197,179.906,5.380,148.966
C01264=1219.895,-52.248,-39.209,179.908,5.381,148.965
C01265=1219.890,-51.998,-39.221,179.911,5.381,148.965
C01266=1219.885,-51.748,-39.233,179.913,5.381,148.964
C01267=1219.880,-51.499,-39.246,179.916,5.381,148.963
C01268=1219.875,-51.249,-39.257,179.918,5.381,148.963
C01269=1219.870,-51.000,-39.270,179.921,5.381,148.962
C01270=1219.865,-50.750,-39.281,179.923,5.382,148.961
C01271=1219.859,-50.501,-39.294,179.925,5.381,148.960
C01272=1219.854,-50.252,-39.307,179.928,5.382,148.960
C01273=1219.849,-50.002,-39.318,179.930,5.382,148.959
C01274=1219.844,-49.752,-39.331,179.933,5.382,148.958
C01275=1219.839,-49.502,-39.343,179.935,5.383,148.958
C01276=1219.834,-49.252,-39.356,179.937,5.382,148.957
C01277=1219.828,-48.983,-39.369,179.940,5.383,148.956
C01278=1219.823,-48.713,-39.382,179.943,5.383,148.956
C01279=1219.817,-48.442,-39.396,179.946,5.383,148.955
C01280=1219.811,-48.173,-39.409,179.948,5.383,148.954
C01281=1219.806,-47.923,-39.421,179.951,5.383,148.953
C01282=1219.801,-47.673,-39.434,179.953,5.383,148.953
C01283=1219.796,-47.424,-39.447,179.955,5.384,148.952
C01284=1219.791,-47.174,-39.458,179.958,5.384,148.951
C01285=1219.786,-46.925,-39.471,179.960,5.384,148.950
C01286=1219.781,-46.675,-39.484,179.963,5.384,148.950
C01287=1219.775,-46.425,-39.496,179.966,5.385,148.949
C01288=1219.771,-46.175,-39.508,179.968,5.384,148.948
C01289=1219.765,-45.926,-39.521,179.970,5.385,148.948
C01290=1219.760,-45.676,-39.533,179.972,5.385,148.947
C01291=1219.755,-45.427,-39.546,179.975,5.385,148.946
C01292=1219.750,-45.178,-39.558,179.977,5.386,148.946
C01293=1219.744,-44.928,-39.570,179.979,5.385,148.945
C01294=1219.740,-44.678,-39.583,179.982,5.386,148.944
C01295=1219.735,-44.428,-39.596,179.985,5.386,148.944
C01296=1219.730,-44.179,-39.608,179.987,5.386,148.943
C01297=1219.724,-43.929,-39.620,179.989,5.387,148.942
C01298=1219.719,-43.680,-39.633,179.991,5.386,148.942
C01299=1219.714,-43.430,-39.646,179.994,5.387,148.941
C01300=1219.709,-43.180,-39.658,179.997,5.387,148.940
C01301=1219.704,-42.930,-39.670,179.999,5.387,148.939
C01302=1219.699,-42.681,-39.683,-179.998,5.387,148.939
C01303=1219.694,-42.432,-39.695,-179.996,5.388,148.938
C01304=1219.688,-42.181,-39.709,-179.994,5.387,148.937
C01305=1219.683,-41.932,-39.721,-179.991,5.388,148.937
C01306=1219.678,-41.682,-39.733,-179.989,5.388,148.936
C01307=1219.673,-41.433,-39.746,-179.986,5.388,148.935
C01308=1219.668,-41.183,-39.759,-179.984,5.389,148.935
C01309=1219.663,-40.934,-39.772,-179.982,5.388,148.934
C01310=1219.658,-40.684,-39.784,-179.979,5.389,148.933
C01311=1219.653,-40.434,-39.796,-179.976,5.389,148.932
C01312=1219.648,-40.184,-39.809,-179.974,5.389,148.932
C01313=1219.642,-39.935,-39.822,-179.971,5.389,148.931
C01314=1219.637,-39.685,-39.835,-179.969,5.390,148.930
C01315=1219.632,-39.436,-39.847,-179.967,5.389,148.930
C01316=1219.627,-39.186,-39.860,-179.964,5.390,148.929
C01317=1219.622,-38.937,-39.873,-179.962,5.390,148.928
C01318=1219.617,-38.687,-39.885,-179.959,5.390,148.928
C01319=1219.612,-38.437,-39.897,-179.957,5.391,148.927
C01320=1219.606,-38.187,-39.911,-179.955,5.390,148.926
C01321=1219.601,-37.938,-39.924,-179.952,5.391,148.926
C01322=1219.596,-37.688,-39.936,-179.950,5.392,148.925
C01323=1219.591,-37.439,-39.949,-179.948,5.391,148.924
C01324=1219.587,-37.189,-39.962,-179.945,5.392,148.924
C01325=1219.581,-36.940,-39.975,-179.942,5.392,148.923
C01326=1219.576,-36.690,-39.988,-179.940,5.392,148.922
C01327=1219.571,-36.440,-40.001,-179.938,5.392,148.921
C01328=1219.566,-36.191,-40.013,-179.935,5.393,148.921
C01329=1219.560,-35.941,-40.026,-179.933,5.393,148.920
C01330=1219.555,-35.692,-40.039,-179.930,5.393,148.919
C01331=1219.550,-35.442,-40.052,-179.928,5.393,148.919
C01332=1219.545,-35.193,-40.065,-179.925,5.393,148.918
C01333=1219.540,-34.943,-40.077,-179.923,5.394,148.917
C01334=1219.535,-34.693,-40.091,-179.921,5.393,148.917
C01335=1219.530,-34.444,-40.103,-179.918,5.394,148.916
C01336=1219.525,-34.194,-40.116,-179.915,5.394,148.915
C01337=1219.519,-33.944,-40.129,-179.913,5.394,148.914
C01338=1219.514,-33.695,-40.142,-179.911,5.395,148.914
C01339=1219.509,-33.445,-40.155,-179.908,5.395,148.913
C01340=1219.505,-33.195,-40.168,-179.906,5.395,148.912
C01341=1219.499,-32.946,-40.181,-179.903,5.395,148.912
C01342=1219.494,-32.696,-40.193,-179.901,5.396,148.911
C01343=1219.489,-32.446,-40.206,-179.898,5.395,148.910
C01344=1219.483,-32.197,-40.220,-179.896,5.396,148.910
C01345=1219.478,-31.947,-40.232,-179.893,5.396,148.909
C01346=1219.474,-31.697,-40.245,-179.891,5.396,148.908
C01347=1219.468,-31.448,-40.258,-179.888,5.396,148.907
C01348=1219.463,-31.198,-40.271,-179.886,5.397,148.907
C01349=1219.458,-30.949,-40.285,-179.884,5.397,148.906
C01350=1219.453,-30.700,-40.297,-179.881,5.397,148.905
C01351=1219.448,-30.449,-40.311,-179.878,5.398,148.905
C01352=1219.443,-30.200,-40.323,-179.876,5.397,148.904
C01353=1219.438,-29.950,-40.336,-179.874,5.398,148.903
C01354=1219.433,-29.700,-40.350,-179.871,5.399,148.903
C01355=1219.427,-29.451,-40.362,-179.869,5.398,148.902
C01356=1219.422,-29.201,-40.376,-179.867,5.399,148.901
C01357=1219.417,-28.952,-40.389,-179.864,5.399,148.901
C01358=1219.413,-28.702,-40.402,-179.862,5.399,148.900
C01359=1219.407,-28.452,-40.415,-179.859,5.399,148.899
C01360=1219.402,-28.203,-40.428,-179.857,5.400,148.899
C01361=1219.398,-27.954,-40.442,-179.855,5.400,148.898
C01362=1219.392,-27.704,-40.455,-179.852,5.400,148.897
C01363=1219.387,-27.454,-40.468,-179.849,5.401,148.897
C01364=1219.381,-27.204,-40.481,-179.847,5.400,148.896
C01365=1219.377,-26.956,-40.494,-179.844,5.401,148.895
C01366=1219.372,-26.706,-40.507,-179.842,5.401,148.894
C01367=1219.366,-26.456,-40.520,-179.840,5.401,148.894
C01368=1219.362,-26.206,-40.533,-179.837,5.401,148.893
C01369=1219.356,-25.957,-40.547,-179.834,5.402,148.892
C01370=1219.352,-25.707,-40.560,-179.832,5.402,148.892
C01371=1219.346,-25.457,-40.573,-179.830,5.402,148.891
C01372=1219.341,-25.207,-40.586,-179.827,5.403,148.890
C01373=1219.336,-24.959,-40.600,-179.824,5.403,148.890
C01374=1219.331,-24.708,-40.613,-179.822,5.403,148.889
C01375=1219.326,-24.459,-40.626,-179.820,5.403,148.888
C01376=1219.320,-24.210,-40.640,-179.817,5.404,148.887
C01377=1219.316,-23.960,-40.653,-179.815,5.403,148.887
C01378=1219.310,-23.710,-40.666,-179.812,5.404,148.886
C01379=1219.306,-23.461,-40.680,-179.810,5.404,148.885
C01380=1219.300,-23.211,-40.693,-179.807,5.404,148.885
C01381=1219.295,-22.942,-40.707,-179.805,5.405,148.884
C01382=1219.289,-22.672,-40.721,-179.802,5.405,148.883
C01383=1219.284,-22.403,-40.736,-179.800,5.406,148.883
C01384=1219.278,-22.134,-40.750,-179.797,5.406,148.882
C01385=1219.274,-21.884,-40.764,-179.795,5.406,148.881
C01386=1219.268,-21.634,-40.777,-179.792,5.406,148.881
C01387=1219.263,-21.385,-40.791,-179.789,5.407,148.880
C01388=1219.258,-21.135,-40.804,-179.787,5.406,148.879
C01389=1219.253,-20.885,-40.817,-179.785,5.407,148.878
C01390=1219.247,-20.636,-40.831,-179.782,5.407,148.878
C01391=1219.243,-20.386,-40.844,-179.779,5.408,148.877
C01392=1219.237,-20.137,-40.858,-179.777,5.408,148.876
C01393=1219.233,-19.887,-40.871,-179.775,5.408,148.876
C01394=1219.227,-19.638,-40.885,-179.772,5.409,148.875
C01395=1219.222,-19.388,-40.898,-179.770,5.408,148.874
C01396=1219.218,-19.139,-40.912,-179.767,5.409,148.874
C01397=1219.212,-18.889,-40.925,-179.765,5.409,148.873
C01398=1219.208,-18.640,-40.939,-179.762,5.410,148.872
C01399=1219.202,-18.390,-40.952,-179.760,5.410,148.871
C01400=1219.197,-18.140,-40.966,-179.757,5.410,148.871
C01401=1219.192,-17.891,-40.979,-179.755,5.411,148.870
C01402=1219.187,-17.641,-40.993,-179.752,5.410,148.869
C01403=1219.182,-17.392,-41.006,-179.750,5.411,148.869
C01404=1219.177,-17.142,-41.020,-179.747,5.411,148.868
C01405=1219.172,-16.892,-41.034,-179.745,5.411,148.867
C01406=1219.167,-16.643,-41.047,-179.742,5.411,148.867
C01407=1219.161,-16.393,-41.061,-179.740,5.412,148.866
C01408=1219.156,-16.144,-41.074,-179.737,5.412,148.865
C01409=1219.151,-15.894,-41.087,-179.735,5.412,148.865
C01410=1219.146,-15.645,-41.101,-179.733,5.413,148.864
C01411=1219.141,-15.395,-41.116,-179.730,5.413,148.863
C01412=1219.136,-15.145,-41.129,-179.728,5.414,148.863
C01413=1219.131,-14.896,-41.142,-179.725,5.414,148.862
C01414=1219.126,-14.646,-41.156,-179.723,5.414,148.861
C01415=1219.121,-14.397,-41.169,-179.720,5.415,148.861
C01416=1219.116,-14.147,-41.184,-179.718,5.414,148.860
C01417=1219.110,-13.897,-41.197,-179.715,5.415,148.859
C01418=1219.106,-13.648,-41.211,-179.713,5.415,148.859
C01419=1219.101,-13.399,-41.225,-179.710,5.416,148.858
C01420=1219.095,-13.148,-41.238,-179.708,5.416,148.857
C01421=1219.091,-12.900,-41.252,-179.705,5.416,148.856
C01422=1219.086,-12.650,-41.266,-179.703,5.417,148.856
C01423=1219.080,-12.400,-41.279,-179.701,5.416,148.855
C01424=1219.075,-12.150,-41.293,-179.698,5.417,148.854
C01425=1219.071,-11.901,-41.307,-179.695,5.417,148.854
C01426=1219.065,-11.651,-41.320,-179.693,5.418,148.853
C01427=1219.060,-11.402,-41.335,-179.691,5.417,148.852
C01428=1219.055,-11.152,-41.349,-179.688,5.418,148.852
C01429=1219.050,-10.903,-41.361,-179.685,5.418,148.851
C01430=1219.045,-10.653,-41.376,-179.683,5.419,148.850
C01431=1219.040,-10.403,-41.390,-179.681,5.419,148.850
C01432=1219.034,-10.154,-41.404,-179.678,5.419,148.849
C01433=1219.030,-9.904,-41.417,-179.675,5.420,148.848
C01434=1219.025,-9.655,-41.431,-179.673,5.420,148.847
C01435=1219.019,-9.406,-41.445,-179.671,5.420,148.847
C01436=1219.014,-9.156,-41.459,-179.668,5.421,148.846
C01437=1219.009,-8.906,-41.474,-179.666,5.421,148.846
C01438=1219.005,-8.656,-41.487,-179.663,5.422,148.845
C01439=1218.999,-8.407,-41.501,-179.661,5.421,148.844
C01440=1218.994,-8.157,-41.515,-179.658,5.422,148.844
C01441=1218.989,-7.908,-41.529,-179.656,5.422,148.843
C01442=1218.984,-7.659,-41.543,-179.653,5.423,148.842
C01443=1218.979,-7.408,-41.557,-179.651,5.423,148.841
C01444=1218.974,-7.159,-41.570,-179.648,5.423,148.841
C01445=1218.969,-6.909,-41.584,-179.646,5.424,148.840
C01446=1218.964,-6.660,-41.598,-179.643,5.424,148.839
C01447=1218.959,-6.411,-41.613,-179.641,5.424,148.839
C01448=1218.954,-6.161,-41.627,-179.638,5.424,148.838
C01449=1218.948,-5.912,-41.641,-179.636,5.425,148.837
C01450=1218.943,-5.662,-41.655,-179.633,5.425,148.837
C01451=1218.939,-5.412,-41.668,-179.631,5.425,148.836
C01452=1218.934,-5.162,-41.682,-179.628,5.426,148.835
C01453=1218.928,-4.913,-41.696,-179.625,5.426,148.835
C01454=1218.923,-4.664,-41.711,-179.623,5.427,148.834
C01455=1218.918,-4.414,-41.725,-179.621,5.426,148.833
C01456=1218.914,-4.164,-41.739,-179.619,5.427,148.833
C01457=1218.908,-3.915,-41.753,-179.616,5.428,148.832
C01458=1218.903,-3.665,-41.767,-179.613,5.428,148.831
C01459=1218.898,-3.416,-41.782,-179.611,5.428,148.831
C01460=1218.893,-3.166,-41.796,-179.609,5.428,148.830
C01461=1218.888,-2.917,-41.809,-179.606,5.429,148.829
C01462=1218.883,-2.668,-41.823,-179.603,5.429,148.829
C01463=1218.878,-2.418,-41.838,-179.601,5.429,148.828
C01464=1218.873,-2.168,-41.852,-179.599,5.430,148.827
C01465=1218.868,-1.919,-41.866,-179.596,5.430,148.826
C01466=1218.863,-1.670,-41.880,-179.593,5.431,148.826
C01467=1218.858,-1.420,-41.894,-179.591,5.431,148.825
C01468=1218.853,-1.170,-41.909,-179.588,5.431,148.824
C01469=1218.848,-0.920,-41.923,-179.586,5.431,148.824
C01470=1218.843,-0.671,-41.937,-179.583,5.432,148.823
C01471=1218.838,-0.422,-41.951,-179.581,5.432,148.822
C01472=1218.833,-0.172,-41.966,-179.578,5.432,148.822
C01473=1218.828,0.078,-41.980,-179.576,5.433,148.821
C01474=1218.823,0.327,-41.994,-179.573,5.433,148.820
C01475=1218.818,0.577,-42.008,-179.571,5.434,148.820
C01476=1218.813,0.827,-42.023,-179.568,5.435,148.819
C01477=1218.807,1.076,-42.037,-179.566,5.434,148.818
C01478=1218.803,1.325,-42.052,-179.564,5.435,148.818
C01479=1218.798,1.575,-42.066,-179.561,5.435,148.817
C01480=1218.793,1.824,-42.080,-179.558,5.436,148.816
C01481=1218.788,2.074,-42.094,-179.556,5.436,148.816
C01482=1218.783,2.324,-42.109,-179.554,5.436,148.815
C01483=1218.777,2.573,-42.123,-179.551,5.437,148.814
C01484=1218.771,2.823,-42.137,-179.548,5.437,148.814
C01485=1218.766,3.092,-42.153,-179.546,5.438,148.813
C01486=1218.761,3.360,-42.169,-179.543,5.438,148.812
C01487=1218.756,3.630,-42.184,-179.540,5.439,148.812
C01488=1218.751,3.899,-42.200,-179.538,5.438,148.811
C01489=1218.746,4.148,-42.214,-179.535,5.438,148.810
C01490=1218.741,4.398,-42.228,-179.533,5.439,148.809
C01491=1218.735,4.647,-42.243,-179.530,5.440,148.809
C01492=1218.730,4.896,-42.258,-179.528,5.440,148.808
C01493=1218.725,5.146,-42.272,-179.526,5.440,148.807
C01494=1218.720,5.396,-42.286,-179.523,5.441,148.807
C01495=1218.715,5.645,-42.301,-179.520,5.441,148.806
C01496=1218.710,5.895,-42.315,-179.518,5.442,148.805
C01497=1218.705,6.144,-42.330,-179.515,5.442,148.805
C01498=1218.700,6.394,-42.344,-179.513,5.442,148.804
C01499=1218.695,6.644,-42.360,-179.510,5.442,148.803
C01500=1218.690,6.893,-42.374,-179.508,5.443,148.803
C01501=1218.685,7.143,-42.388,-179.505,5.443,148.802
C01502=1218.680,7.391,-42.403,-179.502,5.444,148.801
C01503=1218.675,7.641,-42.417,-179.500,5.444,148.801
C01504=1218.670,7.891,-42.431,-179.498,5.444,148.800
C01505=1218.664,8.141,-42.446,-179.495,5.445,148.799
C01506=1218.660,8.390,-42.461,-179.493,5.446,148.799
C01507=1218.655,8.640,-42.475,-179.490,5.446,148.798
C01508=1218.650,8.889,-42.490,-179.487,5.447,148.797
C01509=1218.645,9.138,-42.505,-179.485,5.446,148.797
C01510=1218.639,9.388,-42.520,-179.483,5.447,148.796
C01511=1218.635,9.637,-42.535,-179.480,5.447,148.795
C01512=1218.630,9.887,-42.549,-179.477,5.448,148.795
C01513=1218.625,10.137,-42.563,-179.475,5.448,148.794
C01514=1218.620,10.386,-42.578,-179.473,5.448,148.793
C01515=1218.614,10.636,-42.593,-179.470,5.449,148.793
C01516=1218.610,10.885,-42.608,-179.467,5.449,148.792
C01517=1218.605,11.135,-42.622,-179.465,5.450,148.791
C01518=1218.600,11.385,-42.637,-179.462,5.450,148.791
C01519=1218.594,11.634,-42.652,-179.460,5.451,148.790
C01520=1218.590,11.884,-42.666,-179.458,5.451,148.789
C01521=1218.585,12.133,-42.681,-179.455,5.451,148.789
C01522=1218.580,12.382,-42.696,-179.453,5.452,148.788
C01523=1218.575,12.632,-42.711,-179.450,5.452,148.787
C01524=1218.570,12.882,-42.726,-179.447,5.453,148.787
C01525=1218.565,13.131,-42.741,-179.445,5.453,148.786
C01526=1218.559,13.381,-42.755,-179.443,5.453,148.785
C01527=1218.555,13.630,-42.770,-179.440,5.454,148.785
C01528=1218.550,13.879,-42.785,-179.437,5.454,148.784
C01529=1218.544,14.129,-42.800,-179.435,5.455,148.783
C01530=1218.539,14.379,-42.815,-179.432,5.455,148.783
C01531=1218.535,14.628,-42.830,-179.430,5.455,148.782
C01532=1218.529,14.878,-42.844,-179.428,5.456,148.781
C01533=1218.524,15.127,-42.859,-179.425,5.456,148.781
C01534=1218.519,15.377,-42.874,-179.422,5.457,148.780
C01535=1218.514,15.626,-42.889,-179.420,5.457,148.779
C01536=1218.509,15.876,-42.904,-179.417,5.458,148.779
C01537=1218.504,16.125,-42.919,-179.414,5.459,148.778
C01538=1218.499,16.374,-42.934,-179.412,5.458,148.777
C01539=1218.494,16.624,-42.948,-179.410,5.459,148.777
C01540=1218.489,16.873,-42.963,-179.407,5.459,148.776
C01541=1218.484,17.123,-42.978,-179.404,5.460,148.775
C01542=1218.480,17.373,-42.994,-179.402,5.460,148.775
C01543=1218.474,17.622,-43.009,-179.399,5.461,148.774
C01544=1218.469,17.872,-43.023,-179.398,5.461,148.773
C01545=1218.465,18.121,-43.038,-179.395,5.461,148.773
C01546=1218.459,18.370,-43.054,-179.392,5.462,148.772
C01547=1218.454,18.620,-43.068,-179.390,5.463,148.771
C01548=1218.449,18.869,-43.084,-179.387,5.463,148.771
C01549=1218.444,19.119,-43.099,-179.384,5.464,148.770
C01550=1218.439,19.368,-43.113,-179.382,5.464,148.769
C01551=1218.434,19.618,-43.129,-179.380,5.464,148.769
C01552=1218.429,19.867,-43.144,-179.377,5.464,148.768
C01553=1218.424,20.117,-43.159,-179.374,5.465,148.767
C01554=1218.420,20.367,-43.174,-179.372,5.465,148.767
C01555=1218.414,20.616,-43.190,-179.370,5.466,148.766
C01556=1218.409,20.866,-43.204,-179.367,5.467,148.765
C01557=1218.404,21.115,-43.219,-179.364,5.467,148.765
C01558=1218.399,21.364,-43.234,-179.362,5.467,148.764
C01559=1218.394,21.614,-43.250,-179.360,5.468,148.763
C01560=1218.389,21.863,-43.264,-179.357,5.468,148.763
C01561=1218.384,22.113,-43.280,-179.354,5.469,148.762
C01562=1218.379,22.362,-43.295,-179.352,5.469,148.761
C01563=1218.374,22.612,-43.311,-179.349,5.470,148.761
C01564=1218.369,22.861,-43.326,-179.346,5.470,148.760
C01565=1218.364,23.111,-43.341,-179.344,5.471,148.760
C01566=1218.359,23.360,-43.356,-179.342,5.471,148.759
C01567=1218.354,23.610,-43.372,-179.339,5.471,148.758
C01568=1218.350,23.859,-43.387,-179.337,5.472,148.758
C01569=1218.344,24.109,-43.402,-179.334,5.473,148.757
C01570=1218.340,24.358,-43.417,-179.331,5.473,148.756
C01571=1218.334,24.608,-43.432,-179.329,5.474,148.755
C01572=1218.329,24.857,-43.447,-179.326,5.474,148.755
C01573=1218.324,25.107,-43.463,-179.324,5.475,148.754
C01574=1218.319,25.356,-43.479,-179.321,5.474,148.753
C01575=1218.314,25.605,-43.494,-179.319,5.475,148.753
C01576=1218.309,25.855,-43.509,-179.317,5.476,148.752
C01577=1218.304,26.104,-43.524,-179.314,5.476,148.752
C01578=1218.300,26.354,-43.540,-179.311,5.477,148.751
C01579=1218.294,26.604,-43.555,-179.309,5.477,148.750
C01580=1218.289,26.853,-43.570,-179.306,5.478,148.750
C01581=1218.284,27.103,-43.586,-179.303,5.478,148.749
C01582=1218.280,27.352,-43.601,-179.301,5.479,148.748
C01583=1218.274,27.602,-43.617,-179.299,5.479,148.748
C01584=1218.269,27.851,-43.632,-179.297,5.480,148.747
C01585=1218.264,28.100,-43.647,-179.294,5.480,148.746
C01586=1218.259,28.350,-43.663,-179.291,5.481,148.746
C01587=1218.254,28.600,-43.679,-179.289,5.481,148.745
C01588=1218.250,28.849,-43.694,-179.286,5.482,148.744
C01589=1218.244,29.117,-43.711,-179.283,5.482,148.744
C01590=1218.238,29.386,-43.728,-179.281,5.483,148.743
C01591=1218.233,29.655,-43.743,-179.278,5.483,148.742
C01592=1218.228,29.923,-43.760,-179.275,5.484,148.742
C01593=1218.223,30.173,-43.776,-179.273,5.484,148.741
C01594=1218.218,30.422,-43.791,-179.270,5.485,148.740
C01595=1218.213,30.672,-43.807,-179.267,5.486,148.740
C01596=1218.208,30.921,-43.823,-179.265,5.486,148.739
C01597=1218.203,31.171,-43.839,-179.262,5.487,148.738
C01598=1218.198,31.420,-43.854,-179.260,5.486,148.738
C01599=1218.193,31.670,-43.869,-179.257,5.487,148.737
C01600=1218.188,31.920,-43.885,-179.255,5.488,148.736
C01601=1218.184,32.168,-43.901,-179.253,5.488,148.736
C01602=1218.178,32.418,-43.916,-179.250,5.489,148.735
C01603=1218.173,32.668,-43.932,-179.247,5.489,148.734
C01604=1218.168,32.917,-43.948,-179.245,5.490,148.734
C01605=1218.163,33.166,-43.963,-179.242,5.491,148.733
C01606=1218.158,33.416,-43.978,-179.239,5.491,148.732
C01607=1218.153,33.666,-43.994,-179.237,5.492,148.732
C01608=1218.148,33.915,-44.010,-179.235,5.493,148.731
C01609=1218.143,34.164,-44.026,-179.232,5.493,148.731
C01610=1218.139,34.414,-44.042,-179.230,5.493,148.730
C01611=1218.133,34.663,-44.057,-179.227,5.493,148.729
C01612=1218.128,34.913,-44.073,-179.225,5.494,148.729
C01613=1218.123,35.163,-44.089,-179.222,5.494,148.728
C01614=1218.119,35.411,-44.105,-179.219,5.495,148.727
C01615=1218.113,35.661,-44.120,-179.217,5.496,148.727
C01616=1218.109,35.911,-44.136,-179.215,5.496,148.726
C01617=1218.103,36.160,-44.152,-179.212,5.497,148.725
C01618=1218.098,36.410,-44.168,-179.209,5.497,148.725
C01619=1218.093,36.659,-44.184,-179.207,5.498,148.724
C01620=1218.089,36.908,-44.199,-179.204,5.499,148.723
C01621=1218.084,37.158,-44.215,-179.201,5.499,148.723
C01622=1218.079,37.407,-44.231,-179.199,5.500,148.722
C01623=1218.073,37.656,-44.247,-179.197,5.501,148.722
C01624=1218.069,37.906,-44.263,-179.194,5.501,148.721
C01625=1218.063,38.156,-44.278,-179.192,5.501,148.720
C01626=1218.058,38.405,-44.295,-179.189,5.501,148.720
C01627=1218.054,38.654,-44.310,-179.187,5.502,148.719
C01628=1218.049,38.904,-44.326,-179.184,5.502,148.718
C01629=1218.044,39.153,-44.342,-179.181,5.503,148.718
C01630=1218.039,39.403,-44.358,-179.179,5.504,148.717
C01631=1218.033,39.652,-44.373,-179.177,5.504,148.716
C01632=1218.029,39.902,-44.390,-179.174,5.505,148.716
C01633=1218.024,40.151,-44.406,-179.171,5.506,148.715
C01634=1218.019,40.401,-44.422,-179.169,5.506,148.714
C01635=1218.014,40.650,-44.438,-179.166,5.507,148.714
C01636=1218.009,40.900,-44.454,-179.163,5.507,148.713
C01637=1218.004,41.149,-44.470,-179.161,5.508,148.713
C01638=1217.999,41.398,-44.486,-179.159,5.509,148.712
C01639=1217.994,41.648,-44.501,-179.156,5.509,148.711
C01640=1217.989,41.897,-44.517,-179.153,5.510,148.711
C01641=1217.985,42.147,-44.533,-179.151,5.510,148.710
C01642=1217.980,42.396,-44.550,-179.148,5.511,148.709
C01643=1217.975,42.646,-44.566,-179.146,5.512,148.709
C01644=1217.970,42.894,-44.582,-179.144,5.512,148.708
C01645=1217.965,43.145,-44.598,-179.141,5.512,148.707
C01646=1217.960,43.393,-44.614,-179.138,5.513,148.707
C01647=1217.954,43.643,-44.630,-179.136,5.513,148.706
C01648=1217.950,43.892,-44.646,-179.133,5.514,148.705
C01649=1217.945,44.142,-44.662,-179.131,5.514,148.705
C01650=1217.940,44.391,-44.679,-179.128,5.515,148.704
C01651=1217.935,44.641,-44.694,-179.126,5.516,148.704
C01652=1217.930,44.890,-44.711,-179.123,5.516,148.703
C01653=1217.925,45.139,-44.727,-179.121,5.517,148.702
C01654=1217.920,45.389,-44.743,-179.118,5.517,148.702
C01655=1217.915,45.638,-44.759,-179.115,5.518,148.701
C01656=1217.910,45.888,-44.775,-179.113,5.519,148.701
C01657=1217.904,46.138,-44.792,-179.110,5.519,148.700
C01658=1217.900,46.387,-44.808,-179.108,5.520,148.699
C01659=1217.894,46.636,-44.824,-179.105,5.521,148.699
C01660=1217.890,46.886,-44.841,-179.103,5.521,148.698
C01661=1217.885,47.135,-44.857,-179.100,5.522,148.697
C01662=1217.880,47.385,-44.873,-179.098,5.523,148.697
C01663=1217.876,47.634,-44.889,-179.095,5.523,148.696
C01664=1217.870,47.884,-44.905,-179.092,5.524,148.695
C01665=1217.866,48.133,-44.922,-179.090,5.524,148.695
C01666=1217.861,48.382,-44.938,-179.087,5.525,148.694
C01667=1217.856,48.632,-44.954,-179.085,5.525,148.693
C01668=1217.850,48.881,-44.971,-179.082,5.526,148.693
C01669=1217.846,49.131,-44.988,-179.080,5.527,148.692
C01670=1217.840,49.380,-45.003,-179.077,5.527,148.692
C01671=1217.836,49.630,-45.020,-179.075,5.528,148.691
C01672=1217.831,49.878,-45.036,-179.072,5.528,148.690
C01673=1217.826,50.128,-45.052,-179.069,5.529,148.690
C01674=1217.821,50.378,-45.069,-179.067,5.530,148.689
C01675=1217.816,50.627,-45.085,-179.064,5.530,148.689
C01676=1217.811,50.876,-45.102,-179.062,5.531,148.688
C01677=1217.806,51.126,-45.118,-179.059,5.532,148.687
C01678=1217.801,51.375,-45.135,-179.057,5.532,148.687
C01679=1217.797,51.625,-45.151,-179.054,5.533,148.686
C01680=1217.792,51.874,-45.168,-179.052,5.534,148.685
C01681=1217.786,52.124,-45.184,-179.049,5.534,148.685
C01682=1217.781,52.373,-45.200,-179.046,5.535,148.684
C01683=1217.777,52.622,-45.217,-179.044,5.535,148.683
C01684=1217.772,52.872,-45.234,-179.042,5.536,148.683
C01685=1217.767,53.121,-45.250,-179.039,5.537,148.682
C01686=1217.761,53.371,-45.267,-179.036,5.537,148.682
C01687=1217.756,53.620,-45.283,-179.034,5.538,148.681
C01688=1217.752,53.869,-45.300,-179.031,5.538,148.680
C01689=1217.747,54.119,-45.316,-179.029,5.539,148.680
C01690=1217.742,54.368,-45.333,-179.026,5.540,148.679
C01691=1217.737,54.617,-45.350,-179.024,5.540,148.679
C01692=1217.732,54.867,-45.366,-179.021,5.541,148.678
C01693=1217.727,55.135,-45.383,-179.018,5.542,148.677
C01694=1217.722,55.404,-45.402,-179.016,5.542,148.676
C01695=1217.716,55.672,-45.420,-179.013,5.544,148.676
C01696=1217.711,55.940,-45.437,-179.010,5.544,148.675
C01697=1217.706,56.190,-45.454,-179.007,5.545,148.675
C01698=1217.701,56.440,-45.471,-179.005,5.545,148.674
C01699=1217.696,56.689,-45.487,-179.003,5.546,148.673
C01700=1217.691,56.938,-45.504,-179.000,5.547,148.673
C01701=1217.686,57.188,-45.521,-178.997,5.547,148.672
C01702=1217.681,57.437,-45.537,-178.995,5.548,148.671
C01703=1217.676,57.686,-45.555,-178.992,5.548,148.671
C01704=1217.672,57.936,-45.571,-178.990,5.549,148.670
C01705=1217.667,58.185,-45.588,-178.987,5.550,148.670
C01706=1217.661,58.434,-45.605,-178.985,5.550,148.669
C01707=1217.657,58.684,-45.622,-178.982,5.551,148.668
C01708=1217.652,58.933,-45.638,-178.979,5.552,148.668
C01709=1217.647,59.183,-45.655,-178.977,5.552,148.667
C01710=1217.642,59.432,-45.672,-178.975,5.553,148.667
C01711=1217.638,59.681,-45.688,-178.972,5.554,148.666
C01712=1217.632,59.931,-45.705,-178.969,5.554,148.665
C01713=1217.627,60.180,-45.722,-178.967,5.555,148.665
C01714=1217.622,60.430,-45.739,-178.965,5.556,148.664
C01715=1217.618,60.679,-45.756,-178.962,5.556,148.663
C01716=1217.613,60.928,-45.772,-178.959,5.557,148.663
C01717=1217.607,61.178,-45.790,-178.956,5.558,148.662
C01718=1217.603,61.427,-45.806,-178.954,5.559,148.662
C01719=1217.598,61.677,-45.823,-178.951,5.560,148.661
C01720=1217.593,61.926,-45.840,-178.949,5.560,148.660
C01721=1217.587,62.176,-45.857,-178.946,5.561,148.660
C01722=1217.583,62.425,-45.874,-178.943,5.561,148.659
C01723=1217.579,62.674,-45.891,-178.941,5.562,148.659
C01724=1217.573,62.923,-45.908,-178.939,5.563,148.658
C01725=1217.568,63.173,-45.925,-178.936,5.563,148.657
C01726=1217.563,63.423,-45.942,-178.933,5.564,148.657
C01727=1217.559,63.672,-45.959,-178.931,5.565,148.656
C01728=1217.553,63.920,-45.976,-178.929,5.565,148.655
C01729=1217.549,64.170,-45.993,-178.926,5.566,148.655
C01730=1217.543,64.420,-46.010,-178.923,5.567,148.654
C01731=1217.539,64.669,-46.027,-178.921,5.567,148.653
C01732=1217.534,64.919,-46.044,-178.919,5.568,148.653
C01733=1217.529,65.167,-46.061,-178.916,5.569,148.652
C01734=1217.524,65.417,-46.078,-178.913,5.570,148.652
C01735=1217.519,65.666,-46.095,-178.910,5.571,148.651
C01736=1217.514,65.916,-46.112,-178.908,5.572,148.651
C01737=1217.510,66.166,-46.129,-178.905,5.572,148.650
C01738=1217.505,66.415,-46.147,-178.903,5.573,148.649
C01739=1217.500,66.664,-46.163,-178.900,5.573,148.649
C01740=1217.494,66.913,-46.181,-178.898,5.574,148.648
C01741=1217.489,67.163,-46.198,-178.895,5.575,148.648
C01742=1217.485,67.412,-46.215,-178.893,5.575,148.647
C01743=1217.480,67.662,-46.232,-178.890,5.576,148.646
C01744=1217.475,67.911,-46.249,-178.888,5.577,148.646
C01745=1217.470,68.160,-46.267,-178.885,5.577,148.645
C01746=1217.465,68.409,-46.283,-178.882,5.579,148.644
C01747=1217.460,68.659,-46.301,-178.879,5.579,148.644
C01748=1217.455,68.908,-46.319,-178.877,5.580,148.643
C01749=1217.451,69.158,-46.335,-178.875,5.581,148.643
C01750=1217.446,69.407,-46.353,-178.872,5.581,148.642
C01751=1217.441,69.657,-46.370,-178.869,5.582,148.641
C01752=1217.435,69.906,-46.387,-178.867,5.583,148.641
C01753=1217.431,70.155,-46.405,-178.865,5.584,148.640
C01754=1217.426,70.404,-46.421,-178.862,5.584,148.640
C01755=1217.421,70.654,-46.439,-178.859,5.585,148.639
C01756=1217.416,70.903,-46.457,-178.857,5.586,148.639
C01757=1217.411,71.153,-46.473,-178.854,5.587,148.638
C01758=1217.407,71.402,-46.491,-178.851,5.588,148.637
C01759=1217.401,71.652,-46.509,-178.849,5.588,148.637
C01760=1217.397,71.901,-46.526,-178.847,5.589,148.636
C01761=1217.392,72.150,-46.543,-178.844,5.590,148.636
C01762=1217.386,72.399,-46.561,-178.841,5.590,148.635
C01763=1217.382,72.648,-46.578,-178.839,5.591,148.634
C01764=1217.377,72.897,-46.596,-178.837,5.592,148.634
C01765=1217.372,73.147,-46.613,-178.834,5.592,148.633
C01766=1217.368,73.396,-46.630,-178.831,5.593,148.632
C01767=1217.362,73.646,-46.647,-178.828,5.594,148.632
C01768=1217.358,73.895,-46.665,-178.826,5.595,148.631
C01769=1217.352,74.145,-46.683,-178.823,5.596,148.631
C01770=1217.348,74.394,-46.700,-178.821,5.596,148.630
C01771=1217.343,74.644,-46.717,-178.819,5.597,148.630
C01772=1217.338,74.893,-46.735,-178.816,5.598,148.629
C01773=1217.333,75.143,-46.753,-178.813,5.598,148.628
C01774=1217.329,75.391,-46.770,-178.811,5.599,148.628
C01775=1217.323,75.641,-46.787,-178.808,5.601,148.627
C01776=1217.318,75.890,-46.805,-178.805,5.601,148.627
C01777=1217.314,76.140,-46.823,-178.803,5.602,148.626
C01778=1217.309,76.389,-46.840,-178.800,5.602,148.625
C01779=1217.304,76.638,-46.858,-178.798,5.603,148.625
C01780=1217.299,76.887,-46.876,-178.795,5.604,148.624
C01781=1217.294,77.137,-46.893,-178.793,5.605,148.623
C01782=1217.289,77.386,-46.911,-178.791,5.606,148.623
C01783=1217.285,77.636,-46.928,-178.787,5.607,148.622
C01784=1217.280,77.885,-46.946,-178.785,5.607,148.622
C01785=1217.275,78.134,-46.964,-178.782,5.608,148.621
C01786=1217.270,78.384,-46.981,-178.780,5.609,148.621
C01787=1217.265,78.633,-46.999,-178.777,5.610,148.620
C01788=1217.260,78.882,-47.017,-178.775,5.610,148.619
C01789=1217.256,79.131,-47.034,-178.773,5.611,148.619
C01790=1217.250,79.381,-47.052,-178.769,5.612,148.618
C01791=1217.245,79.630,-47.070,-178.767,5.613,148.618
C01792=1217.241,79.879,-47.088,-178.764,5.614,148.617
C01793=1217.235,80.129,-47.105,-178.762,5.615,148.617
C01794=1217.230,80.378,-47.123,-178.759,5.615,148.616
C01795=1217.226,80.628,-47.141,-178.757,5.616,148.615
C01796=1217.221,80.876,-47.158,-178.755,5.617,148.615
C01797=1217.216,81.145,-47.177,-178.752,5.618,148.614
C01798=1217.211,81.413,-47.196,-178.749,5.619,148.613
C01799=1217.205,81.682,-47.216,-178.746,5.619,148.613
C01800=1217.200,81.950,-47.236,-178.743,5.621,148.612
C01801=1217.196,82.200,-47.252,-178.740,5.621,148.612
C01802=1217.191,82.449,-47.270,-178.738,5.622,148.611
C01803=1217.186,82.698,-47.288,-178.736,5.623,148.610
C01804=1217.181,82.947,-47.306,-178.733,5.623,148.610
C01805=1217.176,83.196,-47.324,-178.730,5.625,148.609
C01806=1217.171,83.446,-47.342,-178.728,5.626,148.609
C01807=1217.166,83.695,-47.360,-178.725,5.626,148.608
C01808=1217.161,83.945,-47.377,-178.722,5.627,148.607
C01809=1217.156,84.194,-47.395,-178.720,5.628,148.607
C01810=1217.151,84.443,-47.413,-178.718,5.628,148.606
C01811=1217.147,84.693,-47.432,-178.715,5.630,148.606
C01812=1217.142,84.942,-47.450,-178.712,5.631,148.605
C01813=1217.137,85.191,-47.468,-178.710,5.631,148.605
C01814=1217.132,85.440,-47.486,-178.707,5.632,148.604
C01815=1217.127,85.690,-47.504,-178.705,5.633,148.604
C01816=1217.122,85.939,-47.522,-178.702,5.633,148.603
C01817=1217.117,86.188,-47.540,-178.699,5.635,148.602
C01818=1217.112,86.437,-47.558,-178.697,5.636,148.602
C01819=1217.108,86.687,-47.576,-178.694,5.636,148.601
C01820=1217.103,86.936,-47.594,-178.692,5.637,148.601
C01821=1217.098,87.185,-47.612,-178.690,5.638,148.600
C01822=1217.093,87.434,-47.630,-178.686,5.639,148.599
C01823=1217.088,87.684,-47.648,-178.684,5.640,148.599
C01824=1217.083,87.933,-47.666,-178.682,5.641,148.598
C01825=1217.078,88.183,-47.685,-178.679,5.641,148.598
C01826=1217.073,88.432,-47.703,-178.676,5.642,148.597
C01827=1217.069,88.681,-47.721,-178.674,5.644,148.597
C01828=1217.064,88.931,-47.739,-178.671,5.644,148.596
C01829=1217.059,89.180,-47.757,-178.669,5.645,148.595
C01830=1217.054,89.429,-47.775,-178.666,5.646,148.595
C01831=1217.050,89.679,-47.793,-178.664,5.646,148.594
C01832=1217.045,89.928,-47.811,-178.661,5.648,148.594
C01833=1217.040,90.177,-47.829,-178.658,5.649,148.593
C01834=1217.035,90.426,-47.847,-178.656,5.649,148.593
